(* CoDeSys 2.3.9.50 project: BallGame_with_PackMLandDriveFB_NT.pro *)
(* Libraries: TcBase.lib 14.5.09 11:14:08, TcSystem.lib 7.6.16 10:01:22, STANDARD.LIB 5.6.98 11:03:02 *)

(* Task configuration *)
TASK BallGame (PRIORITY := 1, INTERVAL := T#10ms);
	PRG_HMI();
	MAIN();
END_TASK
TASK Drive (PRIORITY := 0, INTERVAL := T#5ms);
	PRG_Drive_Link();
END_TASK
TASK Emergency (PRIORITY := 2, INTERVAL := T#5ms);
	PRG_SafetyProgram();
END_TASK

(* Global variable list: Global_Variables *)
VAR_GLOBAL
(* -------------INPUTS and OUTPUTS -------------------*)
(* See Global_Variables_TwinCAT and Global_Variables_CodeSys for
environment specific physical IOs *)

(*-----------------------TIMERS----------------------------*)
	TONMove_Ball_Delay		: TON;
	TONDrive_Delay			: TON;

(*-----------------------COUNTERS----------------------------*)
	CountBallsSortedMetal	: INT:=0;	(*Balls sorted: Metal*)
	CountBallsSortedWooden	: INT:=0;	(*Balls sorted: Wood*)
	CountBallsSortedYellow	: INT:=0;	(*Balls sorted: Wood, Yellow*)
	CountBallsSortedRed		: INT:=0;	(*Balls sorted: Wood, Red*)
	CountBallsSortedBlue	: INT:=0;	(*Balls sorted: Wood, Blue*)
	CountBallsSortedGarbage	: INT:=0;	(*Balls sorted: Unknown*)
	arrCountBallsOnTubes	: ARRAY [1..4] OF INT;	(*Balls on tubes: 1=lower, 2=middle, 3=upper, 4=garbage*)

(*-----------------------FUNCTION BLOCKS----------------*)
	fbDrive					: FB_DriveMovement2;		(*FB for executing the motion*)
	fbStateModel			: FB_StateModel_ST;		(*FB for executing state model*)

(* -------------HMI INPUTS (from HMI to PLC) -------------------*)
	bHMI_BtnStart			: BOOL;		(*Start button on HMI*)
	bHMI_BtnStartLight		: BOOL;		(*Start button Light on HMI*)
	bHMI_BtnStop			: BOOL;		(*Stop button on HMI*)
	bHMI_BtnStopLight		: BOOL;		(*Stop button Light on HMI*)
	bHMI_BtnReset			: BOOL;		(*Reset button on HMI*)
	bHMI_BtnAck		    	: BOOL;		(*Ack button on HMI*)

	HMI_uModeReq			: UINT := 3; (* Default to Sorting

(* -------------HMI OUTPUTS (from PLC to HMI) -------------------*)
	PLC_uModeCurrent		: UINT;		(*Current Mode*)
	PLC_uStateCurrent		: UINT;		(*Current State*)
	O_Light_BeaconRed		: BOOL;		(*Light beacon: Red*)

(*-----------------------OTHER GLOBAL VARS ----------------*)
	bInitCompleted			: BOOL; 	(*Init at Power Up *)
	iBatchSize				: INT := 1;	(*Default Batch Size *)
	iBatchRemaining			: INT;

END_VAR

VAR_GLOBAL CONSTANT
(*-----------------------Lift Position Constants----------------------------*)
	GPOS_LOADING			: WORD := 16#0A;	(*Drive to loading level*)
	GPOS_PIPE_LOW			: WORD := 16#0B;	(*Drive to lower pipe*)
	GPOS_PIPE_MID			: WORD := 16#0C;	(*Drive to middle pipe*)
	GPOS_PIPE_UP			: WORD := 16#0D;	(*Drive to upper pipe*)
	GPOS_GARBAGE			: WORD := 16#0E;	(*Drive to garbage pipe*)
	GPOS_COLOR_SEN			: WORD := 16#0F;	(*Drive to colour sensor*)

(*-----------------------Ball Type Constants----------------------------*)
	METAL					: BOOL := FALSE;
	WOODEN					: BOOL := TRUE;

(*-----------------------TIME Constants----------------------------*)
(*State Model *)
	T_IDLE_SHUTDOWN			: TIME := T#15s;
	T_START_DELAY			: TIME := T#2s;
(*Sorter*)
	T_CLEARING_BALL			: TIME := T#3s;
	T_BALL_DEBOUNCE			: TIME := T#500ms;
	T_LOADING_BALL			: TIME := T#1.5s;	(*Delay for ball to roll from Slot2 to Lifter*)
	T_ROLL_FROM_IND			: TIME := T#500ms;	(*Delay for ball to roll from Slot2 to Lifter*)
	T_REQ_DELAY				: TIME := T#500ms;
(*Drive/Lift*)
	T_RESET_DRIVE_TIME		: TIME := T#500ms;	(*Delay for ball to roll from Slot2 to Lifter*)
	T_DRIVE_DELAY			: TIME := T#2s;	(*Delay for drive to start movement*)
	T_POS_SETTLE_DELAY		: TIME := T#500ms;
	T_EJECTOR_DELAY			: TIME := T#500ms;
	T_COLOUR_SENSOR_DELAY	: TIME := T#1s;
(*Tubes *)
	T_TUBE_EMPTY_DELAY 		: TIME := T#3s;

END_VAR

(* Global variable list: Global_Variables_CodeSys *)
VAR_GLOBAL
(* -------------INPUTS-------------------*)
	ISensorOpt 			:BOOL;	(*Optical sensor - is ball present*)
	ISensorInd 			:BOOL;	(*Inductive sensor - is metal ball present*)
	IEmergencyClear 		:BOOL;	(*Emergency stop is cleared*)
	IRun 				:BOOL;	(*Run switch*)
	ILimitUp 				:BOOL;	(*Lift's limit switch is activated - Up*)
	ILimitLow 		 	:BOOL;	(*Lift's limit switch is activated - Low*)
	IGateClosedMid		:BOOL;	(*Pipe gate closed - Mid*)
	IGateClosedLow		:BOOL;	(*Pipe gate closed - Low*)
	ISorterGateClosed		:BOOL;	(*Sorter gate closed*)
	ISorterLiftUp			:BOOL;	(*Sorter lift at up position*)
	ISorterLiftDown		:BOOL;	(*Sorter lift at down position*)
	IPressureApplied		:BOOL;	(*Pressure is available for the system*)
	TEMP1				:BOOL;
	ISenColourYellow		:BOOL;	(*Colour sensor In1 - Yellow*)
	ISenColourBlue		:BOOL;	(*Colour sensor In2 - Blue*)
	ISenColourGreen		:BOOL;	(*Colour sensor In3 - Green*)
	ISenColourRed		:BOOL;	(*Colour sensor In4 - Red*)
	IDriveStatus 			:WORD;	(*From lift drive status information*)

(* -------------OUTPUTS-------------------*)
	OGateMid			:BOOL;	(*Valve: Open pipe gate - Mid*)
	OGateLow			:BOOL;	(*Valve: Open pipe gate - Low*)
	OSorterGate			:BOOL;	(*Valve: Open sorter gate*)
	OSorterLift			:BOOL;	(*Valve: Sorter lift up*)
	OEjector			:BOOL;	(*Ejector push ball out from lift*)
	ODriveControl 		:WORD;	(*To lift drive control information*)
END_VAR

(* Global variable list: Global_Variables_TwinCAT *)
VAR_GLOBAL
(* -------------INPUTS-------------------*)
	ISensorOpt 			AT %I*	:BOOL;	(*Optical sensor - is ball present*)
	ISensorInd 			AT %I*	:BOOL;	(*Inductive sensor - is metal ball present*)
	IEmergencyClear 	AT %I*	:BOOL;	(*Emergency stop is cleared*)
	IRun 				AT %I*	:BOOL;	(*Run switch*)
	ILimitUp 			AT %I*	:BOOL;	(*Lift's limit switch is activated - Up*)
	ILimitLow 			AT %I* 	:BOOL;	(*Lift's limit switch is activated - Low*)
	IGateClosedUp		AT %I* 	:BOOL;
	IGateClosedMid		AT %I*	:BOOL;	(*Pipe gate closed - Mid*)
	IGateClosedLow		AT %I*	:BOOL;	(*Pipe gate closed - Low*)
	ISorterGateClosed	AT %I*	:BOOL;	(*Sorter gate closed*)
	ISorterLiftUp		AT %I*	:BOOL;	(*Sorter lift at up position*)
	ISorterLiftDown		AT %I*	:BOOL;	(*Sorter lift at down position*)
	IPressureApplied	AT %I*	:BOOL;	(*Pressure is available for the system*)
	TEMP1				AT %I*	:BOOL;
	ISenColourYellow	AT %I*	:BOOL;	(*Colour sensor In1 - Yellow*)
	ISenColourBlue		AT %I*	:BOOL;	(*Colour sensor In2 - Blue*)
	ISenColourGreen		AT %I*	:BOOL;	(*Colour sensor In3 - Green*)
	ISenColourRed		AT %I*	:BOOL;	(*Colour sensor In4 - Red*)
	IDriveStatus 		AT %I*	:WORD;	(*From lift drive status information*)

(* -------------OUTPUTS-------------------*)
	OGateUp				AT %Q*	:BOOL;
	OGateMid			AT %Q*	:BOOL;	(*Valve: Open pipe gate - Mid*)
	OGateLow			AT %Q*	:BOOL;	(*Valve: Open pipe gate - Low*)
	OSorterGate			AT %Q*	:BOOL;	(*Valve: Open sorter gate*)
	OSorterLift			AT %Q*	:BOOL;	(*Valve: Sorter lift up*)
	OEjector			AT %Q*	:BOOL;	(*Ejector push ball out from lift*)
	ODriveControl 		AT %Q*	:WORD;	(*To lift drive control information*)

(* -------------HMI-------------------*)
	I_Btn_Reset		: BOOL;	(*Button: Reset*)
	I_Btn_Start		: BOOL;	(*Button: Start*)
	I_Btn_Stop		: BOOL;	(*Button: Stop*)
	I_Btn_EStop		: BOOL;	(*Button: Reset*)

(* -------------Drive-------------------*)
	bDriveEnabled 	: BOOL;

(* ------------ Manual Mode -------------*)
	bManualMode 	: BOOL := TRUE;
END_VAR

(* Global variable list: TwinCAT_Configuration *)
(* Generated automatically by TwinCAT - (read only) *)
VAR_CONFIG
	.ISensorOpt AT %IX0.0 : BOOL;	(*  ~ {LinkedWith:TIID^Device 4 (EL6731)^Box 2  (BK3110)^Term 2 (KL1002)^Channel 1^Input} *)
	.ISensorInd AT %IX0.1 : BOOL;	(*  ~ {LinkedWith:TIID^Device 4 (EL6731)^Box 2  (BK3110)^Term 2 (KL1002)^Channel 2^Input} *)
	.IEmergencyClear AT %IX0.2 : BOOL;	(*  ~ {LinkedWith:TIID^Device 4 (EL6731)^Box 2  (BK3110)^Term 3 (KL1002)^Channel 1^Input} *)
	.IRun AT %IX0.3 : BOOL;	(*  ~ {LinkedWith:TIID^Device 4 (EL6731)^Box 2  (BK3110)^Term 3 (KL1002)^Channel 2^Input} *)
	.ILimitUp AT %IX0.4 : BOOL;	(*  ~ {LinkedWith:TIID^Device 4 (EL6731)^Box 2  (BK3110)^Term 4 (KL1002)^Channel 1^Input} *)
	.ILimitLow AT %IX0.5 : BOOL;	(*  ~ {LinkedWith:TIID^Device 4 (EL6731)^Box 2  (BK3110)^Term 4 (KL1002)^Channel 2^Input} *)
	.IGateClosedUp AT %IX8.0 : BOOL;
	.IGateClosedMid AT %IX0.7 : BOOL;	(*  ~ {LinkedWith:TIID^Device 4 (EL6731)^Box 2  (BK3110)^Term 5 (KL1104)^Channel 2^Input} *)
	.IGateClosedLow AT %IX1.0 : BOOL;	(*  ~ {LinkedWith:TIID^Device 4 (EL6731)^Box 2  (BK3110)^Term 5 (KL1104)^Channel 3^Input} *)
	.ISorterGateClosed AT %IX1.1 : BOOL;	(*  ~ {LinkedWith:TIID^Device 4 (EL6731)^Box 2  (BK3110)^Term 5 (KL1104)^Channel 4^Input} *)
	.ISorterLiftUp AT %IX1.2 : BOOL;	(*  ~ {LinkedWith:TIID^Device 4 (EL6731)^Box 2  (BK3110)^Term 6 (KL1104)^Channel 1^Input} *)
	.ISorterLiftDown AT %IX1.3 : BOOL;	(*  ~ {LinkedWith:TIID^Device 4 (EL6731)^Box 2  (BK3110)^Term 6 (KL1104)^Channel 2^Input} *)
	.IPressureApplied AT %IX1.4 : BOOL;	(*  ~ {LinkedWith:TIID^Device 4 (EL6731)^Box 2  (BK3110)^Term 6 (KL1104)^Channel 3^Input} *)
	.TEMP1 AT %IX1.5 : BOOL;	(*  ~ {LinkedWith:TIID^Device 4 (EL6731)^Box 2  (BK3110)^Term 6 (KL1104)^Channel 4^Input} *)
	.ISenColourYellow AT %IX1.6 : BOOL;	(*  ~ {LinkedWith:TIID^Device 4 (EL6731)^Box 2  (BK3110)^Term 7 (KL1104)^Channel 1^Input} *)
	.ISenColourBlue AT %IX1.7 : BOOL;	(*  ~ {LinkedWith:TIID^Device 4 (EL6731)^Box 2  (BK3110)^Term 7 (KL1104)^Channel 2^Input} *)
	.ISenColourGreen AT %IX2.0 : BOOL;	(*  ~ {LinkedWith:TIID^Device 4 (EL6731)^Box 2  (BK3110)^Term 7 (KL1104)^Channel 3^Input} *)
	.ISenColourRed AT %IX2.1 : BOOL;	(*  ~ {LinkedWith:TIID^Device 4 (EL6731)^Box 2  (BK3110)^Term 7 (KL1104)^Channel 4^Input} *)
	.IDriveStatus AT %IB4 : WORD;	(*  ~ {LinkedWith:TIID^Device 4 (EL6731)^Box 5 (DKC03)^DKC03 mit LSPM2^Inputs^DKC03 mit LSPM2_0_0} *)
	.OGateUp AT %QX4.0 : BOOL;
	.OGateMid AT %QX0.1 : BOOL;	(*  ~ {LinkedWith:TIID^Device 4 (EL6731)^Box 2  (BK3110)^Term 8 (KL2114)^Channel 2^Output} *)
	.OGateLow AT %QX0.2 : BOOL;	(*  ~ {LinkedWith:TIID^Device 4 (EL6731)^Box 2  (BK3110)^Term 8 (KL2114)^Channel 3^Output} *)
	.OSorterGate AT %QX0.3 : BOOL;	(*  ~ {LinkedWith:TIID^Device 4 (EL6731)^Box 2  (BK3110)^Term 8 (KL2114)^Channel 4^Output} *)
	.OSorterLift AT %QX0.4 : BOOL;	(*  ~ {LinkedWith:TIID^Device 4 (EL6731)^Box 2  (BK3110)^Term 9 (KL2114)^Channel 1^Output} *)
	.OEjector AT %QX0.5 : BOOL;	(*  ~ {LinkedWith:TIID^Device 4 (EL6731)^Box 2  (BK3110)^Term 9 (KL2114)^Channel 2^Output} *)
	.ODriveControl AT %QB2 : WORD;	(*  ~ {LinkedWith:TIID^Device 4 (EL6731)^Box 5 (DKC03)^DKC03 mit LSPM2^Outputs^DKC03 mit LSPM2_1_0} *)
END_VAR

(* Data type *)
TYPE E_BallColour :
(
	NoColour := 0,
	Yellow := 1,
	Blue := 2,
	Red := 3
);
END_TYPE

(* Data type *)
TYPE E_ModeCtrl :
(
	eMode_undefined := 0,
	eMode_Automatic :=1,
	eMode_XXX :=2,
	eMode_Manual :=99,
	eMode_Sorting :=3,
	eMode_Emptying :=4
);
END_TYPE

(* Data type *)
TYPE E_ModeProc :
(*Procedural control modes. Can be changed in any state*)
(
	eModeProc_undefined := 0,
	eModeProc_Automatic :=1,
	eModeProc_SemiAutomatic :=2,
	eModeProc_Manual :=3
);
END_TYPE

(* Data type *)
TYPE E_State :
(
	eSt_Aborting :=0,
	eSt_Aborted,
	eSt_Clearing,
	eSt_Stopped,
	eSt_Stopping,
	eSt_Resetting,
	eSt_Idle,
	eSt_Starting,
	eSt_Execute,
	eSt_Suspending,
	eSt_Suspended,
	eSt_Unsuspending,
	eSt_Holding,
	eSt_Held,
	eSt_UnHolding,
	eSt_Completing,
	eSt_Completed
);
END_TYPE

(* POU PRG_HMI, ST *)
PROGRAM PRG_HMI
VAR_INPUT
	(*HMI Buttons*)
	bBtnResetCounters	: BOOL;	(*Button Reset counters*)
	bBtnEmptyPipes		: BOOL;	(*Button Empty Pipes*)
END_VAR
VAR

	(*Variables for Lift visualisation*)
	iSorterLiftPos	: INT;		(*Position of Sorter Lift cylinder*)
	iLiftPos		: INT;		(*Position of the lift*)
	wTargetPos	: INT;		(*Current target position of the lift*)
	bBall_InLift	: BOOL;		(*Is there a ball in lift*)

	(*internal variables*)
	RS_Ball_InLift	: RS;		(*Flip-flop for ball in the lift*)
	i: INT := 0;		(*Counter*)
	ii: INT := 0;
	SR_EmptyTubes	: SR;


END_VAR
(*Producing blinking signal*)
PRG_Blinking();

(*Sorter lift position calculus*)
IF OSorterLift AND (iSorterLiftPos < 30) THEN
	iSorterLiftPos := iSorterLiftPos +10;
END_IF;
IF NOT OSorterLift AND (iSorterLiftPos > 0) THEN
	iSorterLiftPos := iSorterLiftPos - 10;
END_IF;

(*Lift position calculus*)
CASE fbDrive.wDestination OF
GPOS_PIPE_UP:		(*Go to Pipe Up*)
	wTargetPos:=375;
GPOS_PIPE_MID:	(*Go to Pipe Mid*)
	wTargetPos:=275;
GPOS_COLOR_SEN:	(*Go to Colour sensor*)
	wTargetPos:=220;
GPOS_PIPE_LOW:	(*Go to Pipe Low*)
	wTargetPos:=175;
GPOS_GARBAGE:	(*Go to garbage position*)
	wTargetPos:=110;
GPOS_LOADING:	(*Go to loading position*)
	wTargetPos:=20;
ELSE
	wTargetPos:=0;
END_CASE;

ii := ii + 1;
(*Drive lift*)
IF( ii MOD 3 = 0) THEN
	IF iLiftPos > wTargetPos THEN	(*Lift is higher than target*)
		iLiftPos := iLiftPos - 1;	 (*Go down*)
	ELSIF iLiftPos < wTargetPos THEN	(*Lift is lower than target*)
		iLiftPos := iLiftPos + 1;	 (*Go up*)
	END_IF;
END_IF;

(*Is there a ball in the lift*)
RS_Ball_InLift(
	SET:= (iLiftPos=20 AND OSorterGate),
	RESET1:=OEjector ,
	Q1=>bBall_InLift );

(* ---------------------------------- Button handlers ---------------------------------- *)
(*Button Empty Pipes*)
SR_EmptyTubes (
	SET1:= bBtnEmptyPipes,
	RESET:=,
	Q1=> );
IF SR_EmptyTubes.Q1 THEN
	PRG_EmptyTubes(bExecute:= TRUE, bDone:= );
	SR_EmptyTubes.RESET := FALSE;
	IF PRG_EmptyTubes.bDone THEN
		PRG_EmptyTubes(bExecute:= FALSE);
		SR_EmptyTubes.RESET := TRUE;
	END_IF
END_IF

(*Button Reset coutners*)
IF bBtnResetCounters THEN
	CountBallsSortedMetal := 0;
	CountBallsSortedWooden := 0;
	CountBallsSortedYellow := 0;
	CountBallsSortedBlue := 0;
	CountBallsSortedRed := 0;
	CountBallsSortedGarbage := 0;
	FOR i := 1 TO 3 DO
		arrCountBallsOnTubes[i] := 0;
	END_FOR;
END_IF;
END_PROGRAM

(* POU Background Programs/PRG_Blinking, ST *)
PROGRAM PRG_Blinking
(*Supporting caluculations: Blinking signals
Author: 	Niko Siltala, niko.siltala@tut.fi
Date: 	2014-01-01*)

VAR_OUTPUT
	bSign4Hz	:BOOL;				(*4 Hz (240krt/min) taajudella vaihteleva signaali*)
	bSign2Hz	:BOOL;				(*2 Hz (120krt/min) taajudella vaihteleva signaali*)
	bSign1Hz	:BOOL;				(*1 Hz (60krt/min) taajudella vaihteleva signaali*)
	bSign0_5Hz	:BOOL;				(*0,5 Hz (30krt/min) taajudella vaihteleva signaali*)
END_VAR
VAR
	bInitDone	: BOOL	:=FALSE;		(*Ohjelman initialisointi*)
	TP_Delay	: TP;					(*Nopein taajuus / 2 tuottaja*)
	bBaseHz	: BOOL	:=FALSE;		(*Nopein taajuus/2*)
	iBaseHz		: UINT	:=4;			(*Base taajuus (Hz)*)
	RTRIG_2Hz_Sign 	: R_TRIG;		(*2Hz signaalin generointi*)
	RTRIG_1Hz_Sign 	: R_TRIG;		(*1Hz signaalin generointi*)
	RTRIG_0_5Hz_Sign	: R_TRIG;	(*0,5Hz signaalin generointi*)
	tBaseTaajuus	:TIME;			(*Base vilkutuksen timerin arvo. f/2*)
	fPLC_CYCLE_TIME	: LREAL;		(*PLC:n cycli aika. Sekunttia*)
END_VAR
(*Ohjelman initialisoinnit - Suoritetaan vain kertaalleen*)
IF NOT bInitDone THEN
	fPLC_CYCLE_TIME := UDINT_TO_LREAL(SystemTaskInfoArr[1].cycleTime) / 10E6;
	(*Base Vilkkusignaalien tuottaminen*)
	(* 250ms - 1* cykliaika(20ms)*)
	tBaseTaajuus := LREAL_TO_TIME( ( (1/ UINT_TO_LREAL(iBaseHz) / 2 ) - 1 * fPLC_CYCLE_TIME ) * 1000);
	bInitDone := TRUE;
END_IF;


(*Base signaalin genrointi*)
TP_Delay(IN:=NOT TP_Delay.Q , PT:=tBaseTaajuus);
IF NOT TP_Delay.Q THEN
	bBaseHz := NOT bBaseHz;
	bSign4Hz:= bBaseHz;
END_IF;

(*2Hz signaalin genrointi*)
RTRIG_2Hz_Sign(CLK:=bSign4Hz);
IF RTRIG_2Hz_Sign.Q THEN
	bSign2Hz:=NOT bSign2Hz;
END_IF;

(*1Hz signaalin genrointi*)
RTRIG_1Hz_Sign(CLK:=bSign2Hz);
IF RTRIG_1Hz_Sign.Q THEN
	bSign1Hz:=NOT bSign1Hz;
END_IF;

(*0,5 Hz signaalin generointi*)
RTRIG_0_5Hz_Sign(CLK:=bSign1Hz);
IF (RTRIG_0_5Hz_Sign.Q) THEN
	bSign0_5Hz:= NOT bSign0_5Hz;
END_IF;
END_PROGRAM

(* POU Processes/PRG_EmptyTubes, SFC *)
(* This Program performs the emptying of the tubes in a set sequence
to prevent jamming. Used in User mode: Emptying
Author: Nicolas Trimborn, nicolas.trimborn@tuni.fi
Date: 	2020-03-01*)

PROGRAM PRG_EmptyTubes
VAR_INPUT
	bExecute	: BOOL;
END_VAR
VAR_INPUT
	bDone		: BOOL;
	bStopOk		: BOOL;
END_VAR
VAR
	fbDelay		:FB_Wait;
END_VAR
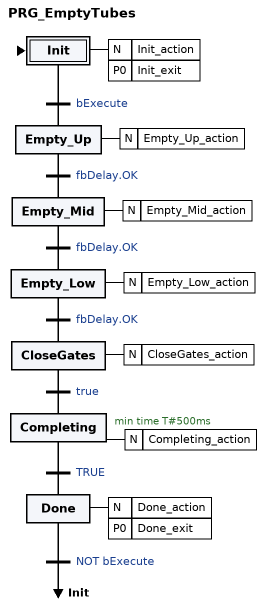
INITIAL_STEP Init:
	Init_action(N);
	Init_exit(P0);
END_STEP
TRANSITION FROM Init TO Empty_Up := bExecute;
END_TRANSITION
STEP Empty_Up:
	Empty_Up_action(N);
END_STEP
TRANSITION FROM Empty_Up TO Empty_Mid := fbDelay.OK;
END_TRANSITION
STEP Empty_Mid:
	Empty_Mid_action(N);
END_STEP
TRANSITION FROM Empty_Mid TO Empty_Low := fbDelay.OK;
END_TRANSITION
STEP Empty_Low:
	Empty_Low_action(N);
END_STEP
TRANSITION FROM Empty_Low TO CloseGates := fbDelay.OK;
END_TRANSITION
STEP CloseGates:
	CloseGates_action(N);
END_STEP
TRANSITION FROM CloseGates TO Completing := true;
END_TRANSITION
STEP Completing: (* min time T#500ms *)
	Completing_action(N);
END_STEP
TRANSITION FROM Completing TO Done := TRUE;
END_TRANSITION
STEP Done:
	Done_action(N);
	Done_exit(P0);
END_STEP
TRANSITION FROM Done TO Init := NOT bExecute;
END_TRANSITION

ACTION Init_action:
bStopOk := TRUE;
END_ACTION

ACTION Init_exit:
(* Sequence is executing, Reset progress flags *)
bDone 	:= FALSE;
bStopOk := FALSE;
END_ACTION

ACTION Empty_Up_action:
fbDelay(IN_TIME:=T_TUBE_EMPTY_DELAY);
OGateUp := TRUE;
END_ACTION

ACTION Empty_Mid_action:
fbDelay(IN_TIME:=T_TUBE_EMPTY_DELAY);
OGateMid := TRUE;
END_ACTION

ACTION Empty_Low_action:
fbDelay(IN_TIME:=T_TUBE_EMPTY_DELAY);
OGateLow := TRUE;
END_ACTION

ACTION CloseGates_action:
OGateLow := FALSE;
OGateMid := FALSE;
OGateUp  := FALSE;
END_ACTION

ACTION Completing_action:
fbStateModel.bComplete := TRUE;
END_ACTION

ACTION Done_action:
(* Sequence Completed, set progress flags *)
bDone := TRUE;
bStopOk := TRUE;
fbStateModel.bSC := TRUE;
END_ACTION

ACTION Done_exit:
bDone := FALSE;
END_ACTION
END_PROGRAM

(* POU FBs/FB_Wait, ST *)
FUNCTION_BLOCK FB_Wait
(*Waits the given time and sets output after timer has run till end. When called again timer restarts.
Author: 	Niko Siltala, niko.siltala@tut.fi
Date: 	2014-01-01*)
VAR_INPUT
	IN_TIME	:TIME;		(*Time to wait*)
END_VAR
VAR_OUTPUT
	OK 		: BOOL:=FALSE;	(*Gets true after wait time has expired*)
END_VAR
VAR
	Timer	: TP;
	Falling	: F_TRIG;
END_VAR
IF Timer.Q=TRUE THEN
	(*Call timer block when pulse timer is counting*)
	Timer;
ELSE
	(*Timer has espired. Start it again*)
	Timer(IN:=FALSE);
	Timer(PT:=IN_TIME);
	Timer(IN:=TRUE);
END_IF;
(*Set output. True if timer has expired*)
OK:=NOT Timer.Q;
END_FUNCTION_BLOCK

(* POU MAIN, ST *)
(* Main performs Implements PackML model to control the execution of the application
used to coordinate machine operation. 
User modes are:
 - Sorting
 - Emptying
PRG_Safety is running as a separate process to monitor the Estop and limit switches
to shut down drive regardless of other program logic.
Author: Nicolas Trimborn, nicolas.trimborn@tuni.fi
Date: 	2020-03-01*)

PROGRAM MAIN

VAR
	runTrigger			: R_TRIG;
	stopTrigger			: F_TRIG;
	tonStarting			: TON;	(* Start timer used to provide notification machine is starting *)
	rsEmergencyClear	: RS;	(*RS - flip-flop for Emergency clear info*)
	fbPipeUp    		: FB_Pipe;
	fbPipeMid   		: FB_Pipe;
	fbPipeLow   		: FB_Pipe;
	fbDelay				: FB_Wait;
END_VAR
(* ****** Section 1: Initialisations and default values. Initial conditions for variables on every PLC cycle*)
(*Default values*)
fbStateModel.bSC := FALSE;
runTrigger(CLK := IRun); (* finds the counting up events *)
stopTrigger(CLK := IRun); (* finds the clear commands *)

(*System resets*)

(* ****** Section 2: Actions in your program without considering the Control Mode. I.e. actions are performed same way indenpendent on
current Control Mode selection.*)
(*Mode independent state actions. Change / Add / Remove states according your need*)
CASE fbStateModel.eState OF
	eSt_Aborting: (* Handles aborting action such as E-Stop, Limit Switches and Pressure loss *)
		actAborting;
		fbStateModel.bSC := TRUE;		(*MODIFY*)
	eSt_Clearing:
		fbDrive(bReset := TRUE);
		fbDelay(IN_TIME:= T_RESET_DRIVE_TIME, OK=> );
		IF fbDelay.OK THEN
			fbDrive(bReset := FALSE);
			fbStateModel.bSC := TRUE;
		END_IF
	eSt_Resetting:
		tonStarting(IN:=FALSE , PT:= , Q=> , ET=> );	(*MODIFY*)
		fbStateModel.bComplete  := FALSE;
		fbStateModel.bSC := TRUE;
	eSt_Starting:
		(* Reset Program Reset Flags *)
		PRG_Initialisation(bReset := FALSE);
		PRG_Sorting.bReset := FALSE;
		PRG_HMI.bBtnResetCounters := FALSE;
		(* Starting Sequence,  Need to check that pressure is avalible and emergency is clear *)
		IF NOT bInitCompleted THEN (* Initial Startup - Perform Initialisation *)
			PRG_Initialisation(bExecute:= TRUE, bReset := FALSE );
		ELSE (* Init Not Required, Start after 2s delay *)
			fbDrive(bEnable:= TRUE, bStart := TRUE);
			IF fbDrive.bHomingDone THEN
				tonStarting(IN:=TRUE , PT:=T_START_DELAY , Q=> , ET=> );
				IF tonStarting.Q THEN
					fbStateModel.bSC := TRUE;
				END_IF
			END_IF
		END_IF
	
		IF PRG_Initialisation.bDone THEN (*Initialisation Program Is Done *)
			(*Reset Init Program and set bInitComplete flag to indicate Init Performed on Power Up*)
			PRG_Initialisation(bReset:= , bExecute:= FALSE , bDone=> );
			bInitCompleted := TRUE;
		END_IF
	eSt_Holding:
		fbStateModel.bSC := TRUE;		(*MODIFY*)
	eSt_UnHolding:
		fbStateModel.bSC := TRUE;		(*MODIFY*)
	eSt_Suspending:
		fbStateModel.bSC := TRUE;		(*MODIFY*)
	eSt_Unsuspending:
		fbStateModel.bSC := TRUE;		(*MODIFY*)
END_CASE;

(* ****** Section 3: Actions in your program which are Control Mode specific. Two nested case structures where outer one selects the
control mode and inner the PackML state. In order to avoid conflicts, it would be better to process each PackML state either in Section 2 
or Section 3, but not in both. *)
(*Execution mode related state actions. Change / Add / Remove mode and states according your need*)
CASE fbStateModel.eMode OF
	(* ********************* MODE: Emptying******************************************************* *)
	eMode_Emptying:
		(* ****** Section 3.1: PackML state based processing actions when Control Mode is Emptying.*)
		CASE fbStateModel.eState OF
			eSt_Stopping: (*Ensure sequence completeded before stopping, Nice Stop*)
				PRG_EmptyTubes(bExecute:= FALSE, bDone:= , bStopOk:= );
				IF PRG_EmptyTubes.bStopOk THEN
					fbStateModel.bSC := TRUE;
				END_IF
			eSt_Completed:
				fbStateModel.bComplete  := FALSE;
				PRG_EmptyTubes(bExecute := FALSE);
				PRG_HMI.bBtnResetCounters := TRUE;
		END_CASE;

		IF  (fbStateModel.eState>eSt_Starting) AND (fbStateModel.eState<=eSt_Completing) THEN (*State is equal or above Stopped*)
			(*Make here the actions / calls Good place to start with is PRG_Sorting (PRG)*)
			PRG_EmptyTubes(bExecute:= TRUE, bDone:= , bStopOk:= );

		END_IF;

	(* ********************* MODE: Manual ******************************************************* *)
	eMode_Manual:
		CASE fbStateModel.eState OF
		eSt_Stopping:
			;
		eSt_Execute:
			;
		END_CASE;


	(* ********************* MODE: Sorting ****************************************************** *)
	eMode_Sorting:
		(* ****** Section 3.2: PackML state based processing actions when Control Mode is Sorting.*)
		CASE fbStateModel.eState OF
		(*
		eSt_Idle:
			(* Reset Start Counter and bComplete Flag
			tonStarting(IN:=FALSE , PT:= , Q=> , ET=> );
			fbStateModel.bComplete  := FALSE;
			fbStateModel.bSC 		:= TRUE; *)
		eSt_Stopping:
			PRG_Sorting(bExecute:= FALSE, bDone:= , bStopOk:= );
			IF PRG_Sorting.bStopOk THEN
				fbStateModel.bSC := TRUE;
			END_IF
		eSt_Completed:
			fbStateModel.bComplete := FALSE;
			IF fbStateModel.bAck_Completed OR bHMI_BtnAck THEN
				PRG_HMI.bBtnResetCounters := TRUE;
				PRG_Sorting.bReset := TRUE;
			END_IF
			;
		END_CASE; (*fbStateModel.eState *)

	(* ****** Section 4: Grouping PackML states for calling Programs or FB instances.
	This is to avoid repetition inside above case structure in Section 3. With IF clause setting lower (and upper) state limits we can filter out the states when we want to call 
	specific programs. The order of states is defined in Tab:Data types > E_PackMLState. eSt_Aborting is lowest and eSt_Completed is highest.
	Here we filter calling programs, only when we are in higher states than Stopped. 
	This can be pulled out as completely separated section, like in PackML_StateModel_v2-2.pro project. There is inside IF again CASE which process each Control Mode separately.*)
	(*Execution part. Making calls for program if we are on states above Stopped*)
		(*If we are between specific states, make some action or program call*)
			(*IF  (fbStateModel.eState>eSt_Starting) AND (fbStateModel.eState<=eSt_Completing) THEN*)
		IF  (fbStateModel.eState>eSt_Starting) AND (fbStateModel.eState<=eSt_Completing) THEN (*State is equal or above Stopped*)
			(*Make here the actions / calls Good place to start with is PRG_Sorting (PRG)*)
			PRG_Sorting(bExecute:= TRUE , bReset:= , bDone=> , bStopOk=>, iBatchSize := iBatchSize );
		END_IF;

	(* ********************* End of MODE: Sorting******************************************************* *)


	(* fbStateModel.eMode, MODE: UNKNOWN*)
	ELSE	(*Error*)
		; (*TODO*)
END_CASE;

(* ****** Section 5: Calling the fbStateModel instance.
Here the instance of state model is called and all triggering inputs are set, but bSC (State Completed), which you control in your programs. 
This is indication that your program has  finished certain stage.
- Pay attention where the instance fbStateModel is defined. Do you do it in global variables or e.g. here in PRG_MAIN? Important is to use the 
same instance in all places, so that machine state is unique and shared. Remember, if you have multiple definitions, the PRG_MAIN "hides" 
the global one, and might lead to problems elswhere, when you think you are using the same instance, but actually are not. 
- In case you are using the PackML visualisation (VC_PackMLStates), make sure you connect its placeholder to the very same PackML FB instance.
- The Mask for wIgnoreState is created as following. I use binary base for the value(2#). The lowest bit in the mask corresponds the eSt_Aborting
 in E_PackMLState. The next is eSt_Aborted, and so on. Specific state is ignored and jumped over when it is masked out i.e. ignored by having 1 
in that position. Note that implementation allows this only for selected states. See FB_PackMLStateModel_ST code for further details.*)
(*Calling & Updating the state model*)
(*TODO: Evaluate and change all input conditions according your application needs*)
fbStateModel(
	bResetFB:= ,
	eModeReq:= HMI_uModeReq,
	wIgnoreState := 2#1000000,		(*TODO: Which states should be ignodered. Default: 2#000000 or 2#100000. The latter is ignoring Resetting state*)
	bSC:= ,			(*Must not be assigned ANY variable, because fb input is directly operated!!!*)
	bAbort:= NOT IEmergencyClear OR NOT IPressureApplied OR ILimitLow OR ILimitUp,
	bClear:= IEmergencyClear,
	bReset:= runTrigger.Q OR bHMI_BtnReset OR bHMI_BtnStart,
	bStart:= runTrigger.Q OR bHMI_BtnStart,
	bHold:= ,
	bUn_Hold:= ,
	bSuspend:= ,
	bUn_Suspend:= ,
	bStop:= bHMI_BtnStop OR stopTrigger.Q,
	bComplete:= ,
	bAck_Completed:= bHMI_BtnAck OR bHMI_BtnReset ,
	eMode=> PLC_uModeCurrent,
	eState=> PLC_uStateCurrent);

(* ****** Section 6: Here we update all outputs according the current state of our PackML model. This allows us to process the in single location.
The control of outputs is bind to state, not e.g. to inputs. The inputs are the one driving the PackML model forward. Again CASE structure can be used.*)
(*Call for HMI and UI update*)
(*PRG_Drive_Link()*);
HMI_and_UI_Update;
END_PROGRAM
ACTION actAborting:
(*PRG_Sorting(bReset:=TRUE , bExecute:= FALSE);*)
(*bInitCompleted := FALSE;*)
fbDrive(bEnable:= FALSE );
;
END_ACTION
ACTION HMI_and_UI_Update:
(*Simulate emergency stop circuitry
rsEmergencyClear(
	SET:= I_Btn_Reset,
	RESET1:= I_Btn_EStop ,
	Q1=> IEmergencyClear);
*)

(*HMI Update*)
PRG_Blinking (bSign4Hz=> , bSign2Hz=> , bSign1Hz=> , bSign0_5Hz=> );
PRG_Sorting.actCountBallsProcessed;
(*iBatchRemaining := iBatchSize - PRG_AutoSort.iBallsProcessed;*)

(*Init values*)
O_Light_BeaconRed := FALSE;
fbPipeLow(str_PipeName:= 'Metal', i_arrCountBallsIndex := 1, I_GateClosed := IGateClosedLow );
fbPipeMid(str_PipeName:= 'Wood, Blue' , i_arrCountBallsIndex := 2, I_GateClosed := IGateClosedMid );
fbPipeUp(str_PipeName:= 'Wood, Yellow', i_arrCountBallsIndex := 3, I_GateClosed := IGateClosedUp );

(*OLight_Start :=  (fbStateModel.eState >= eSt_Resetting) AND (fbStateModel.eState < eSt_Completed);*)
CASE fbStateModel.eState OF
eSt_Aborting, eSt_Aborted:
	O_Light_BeaconRed := PRG_Blinking.bSign1Hz;
	bHMI_BtnStartLight:= FALSE;
	bHMI_BtnStopLight := PRG_Blinking.bSign1Hz;
eSt_Clearing:
	O_Light_BeaconRed := PRG_Blinking.bSign0_5Hz;
	bHMI_BtnStopLight := PRG_Blinking.bSign0_5Hz;
eSt_Stopped, eSt_Completed:
	O_Light_BeaconRed := TRUE;
	bHMI_BtnStartLight:= FALSE;
	bHMI_BtnStopLight := TRUE;
eSt_Starting:
	bHMI_BtnStartLight := PRG_Blinking.bSign0_5Hz;
	bHMI_BtnStopLight := FALSE;
eSt_Stopping:
	bHMI_BtnStartLight := PRG_Blinking.bSign1Hz;
	bHMI_BtnStopLight := TRUE;
eSt_Execute:
	bHMI_BtnStartLight := TRUE;
	bHMI_BtnStopLight := FALSE;
	;
END_CASE;
END_ACTION

(* POU FBs/FB_Pipe, SFC *)
FUNCTION_BLOCK FB_Pipe
VAR_INPUT
	bReset					: BOOL;	(*Reset Request*)
	str_PipeName			: STRING;
	i_arrCountBallsIndex	: INT;
	I_GateClosed			: BOOL;
END_VAR
VAR_OUTPUT

END_VAR
VAR
	iBallCount  : INT := 0;
	tBallDelay	: TIME := T#1s;
	fbDelay		: FB_Wait;
	bLocalReset	: BOOL;	(*Performs local reset*)
	SFCReset 	: BOOL;	(*Resets the execution of SFC to init once this SFCFlag is set true *)
END_VAR
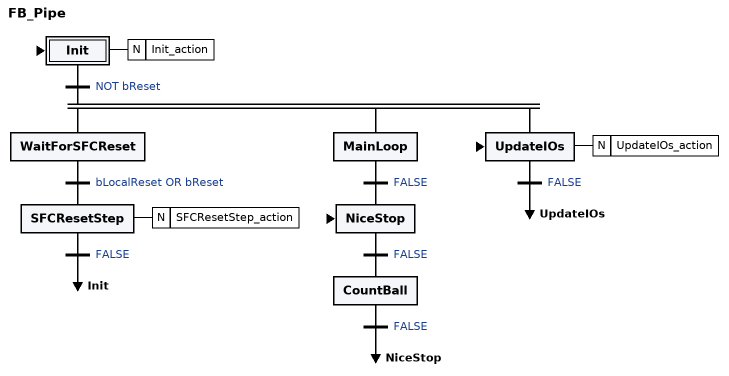
INITIAL_STEP Init:
	Init_action(N);
END_STEP
TRANSITION FROM Init TO (WaitForSFCReset, MainLoop, UpdateIOs) := NOT bReset;
END_TRANSITION
STEP WaitForSFCReset:
END_STEP
TRANSITION FROM WaitForSFCReset TO SFCResetStep := bLocalReset OR bReset;
END_TRANSITION
STEP MainLoop:
END_STEP
TRANSITION FROM MainLoop TO NiceStop := FALSE;
END_TRANSITION
STEP NiceStop:
END_STEP
TRANSITION FROM NiceStop TO CountBall := FALSE;
END_TRANSITION
STEP CountBall:
END_STEP
TRANSITION FROM CountBall TO NiceStop := FALSE;
END_TRANSITION
STEP UpdateIOs:
	UpdateIOs_action(N);
END_STEP
TRANSITION FROM UpdateIOs TO UpdateIOs := FALSE;
END_TRANSITION
STEP SFCResetStep:
	SFCResetStep_action(N);
END_STEP
TRANSITION FROM SFCResetStep TO Init := FALSE;
END_TRANSITION

ACTION Init_action:
SFCReset := FALSE;
bLocalReset	:= FALSE;
END_ACTION

ACTION UpdateIOs_action:
iBallCount := arrCountBallsOnTubes[i_arrCountBallsIndex];
END_ACTION

ACTION SFCResetStep_action:
SFCReset := TRUE;
END_ACTION
END_FUNCTION_BLOCK

(* POU Processes/PRG_Initialisation, SFC *)
(* This Program performs the initialising of the sorting machine to ensure it
enters a know state before sorting begins.  
- Clears sorter lift to ensure any balls left drop to lift
- Close Pipe Gates
- Home Lift and take any balls to garbage chute before returning to loading pos.
Author: Nicolas Trimborn, nicolas.trimborn@tuni.fi
Date: 	2020-03-01*)

PROGRAM PRG_Initialisation
(*Template program for system initialisation*)
VAR_INPUT
	bReset			: BOOL := FALSE;(*Reseting the SFC*)
	bExecute		: BOOL;			(*Executes PRG*)
END_VAR
VAR_OUTPUT
	bDone			: BOOL;			(*Program operations done*)
END_VAR
VAR
(* -------------INTERNAL-------------------*)
	tonMoveDelay	: TON;
	tonBallClearing	: TON;
	fbDelay			: FB_Wait;

	bSorterLiftClear: BOOL:=FALSE;
	bGatesClosed	: BOOL:=FALSE;
	bActuRetracted	: BOOL:=FALSE;
	bDriveAtLoading	: BOOL:=FALSE;
	bDriveReady		: BOOL:=FALSE;

(*System variables. See SFC-flags: http://infosys.beckhoff.com/content/1033/tcplccontrol/html/tcplcctrl_editorsfc.htm?id=24319#SFC-Flags*)
	SFCReset		: BOOL := FALSE;	(*For reseting the SFC*)
END_VAR
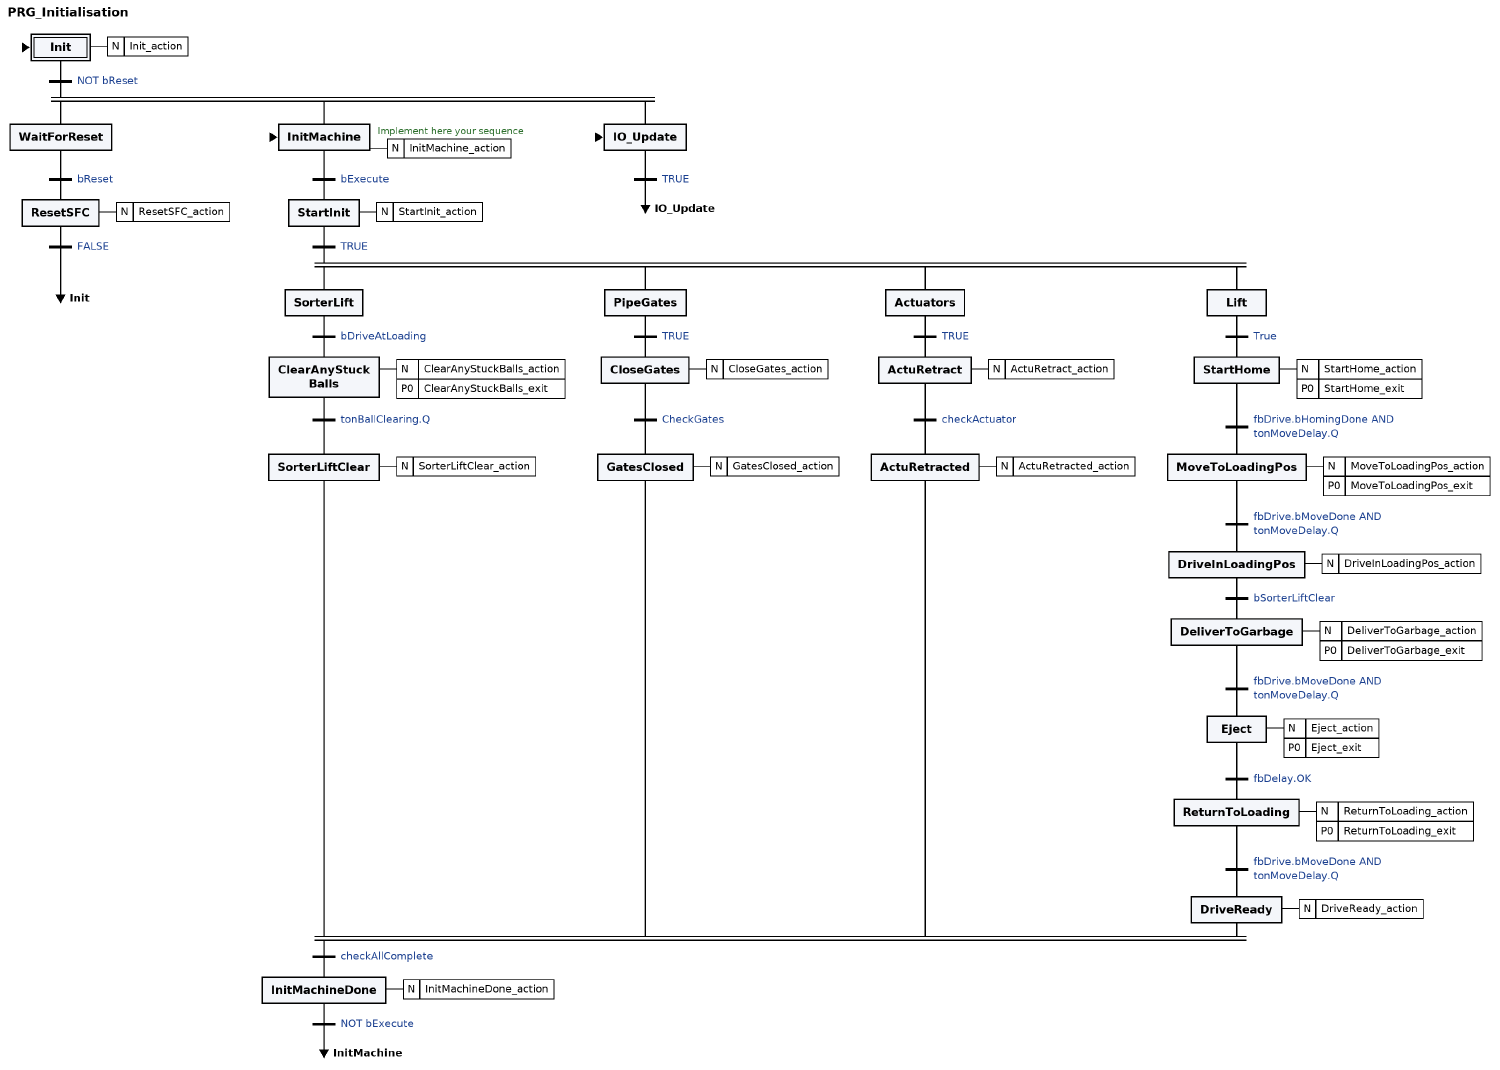
INITIAL_STEP Init:
	Init_action(N);
END_STEP
TRANSITION FROM Init TO (WaitForReset, InitMachine, IO_Update) := NOT bReset;
END_TRANSITION
STEP WaitForReset:
END_STEP
TRANSITION FROM WaitForReset TO ResetSFC := bReset;
END_TRANSITION
STEP InitMachine: (* Implement here your sequence *)
	InitMachine_action(N);
END_STEP
TRANSITION FROM InitMachine TO StartInit := bExecute;
END_TRANSITION
STEP StartInit:
	StartInit_action(N);
END_STEP
TRANSITION FROM StartInit TO (SorterLift, PipeGates, Actuators, Lift) := TRUE;
END_TRANSITION
STEP SorterLift:
END_STEP
TRANSITION FROM SorterLift TO ClearAnyStuckBalls := bDriveAtLoading;
END_TRANSITION
STEP ClearAnyStuckBalls:
	ClearAnyStuckBalls_action(N);
	ClearAnyStuckBalls_exit(P0);
END_STEP
TRANSITION FROM ClearAnyStuckBalls TO SorterLiftClear := tonBallClearing.Q;
END_TRANSITION
STEP SorterLiftClear:
	SorterLiftClear_action(N);
END_STEP
STEP PipeGates:
END_STEP
TRANSITION FROM PipeGates TO CloseGates := TRUE;
END_TRANSITION
STEP CloseGates:
	CloseGates_action(N);
END_STEP
TRANSITION FROM CloseGates TO GatesClosed := CheckGates;
END_TRANSITION
STEP GatesClosed:
	GatesClosed_action(N);
END_STEP
STEP Actuators:
END_STEP
TRANSITION FROM Actuators TO ActuRetract := TRUE;
END_TRANSITION
STEP ActuRetract:
	ActuRetract_action(N);
END_STEP
TRANSITION FROM ActuRetract TO ActuRetracted := checkActuator;
END_TRANSITION
STEP ActuRetracted:
	ActuRetracted_action(N);
END_STEP
STEP Lift:
END_STEP
TRANSITION FROM Lift TO StartHome := True;
END_TRANSITION
STEP StartHome:
	StartHome_action(N);
	StartHome_exit(P0);
END_STEP
TRANSITION FROM StartHome TO MoveToLoadingPos := fbDrive.bHomingDone AND tonMoveDelay.Q;
END_TRANSITION
STEP MoveToLoadingPos:
	MoveToLoadingPos_action(N);
	MoveToLoadingPos_exit(P0);
END_STEP
TRANSITION FROM MoveToLoadingPos TO DriveInLoadingPos := fbDrive.bMoveDone AND tonMoveDelay.Q;
END_TRANSITION
STEP DriveInLoadingPos:
	DriveInLoadingPos_action(N);
END_STEP
TRANSITION FROM DriveInLoadingPos TO DeliverToGarbage := bSorterLiftClear;
END_TRANSITION
STEP DeliverToGarbage:
	DeliverToGarbage_action(N);
	DeliverToGarbage_exit(P0);
END_STEP
TRANSITION FROM DeliverToGarbage TO Eject := fbDrive.bMoveDone AND tonMoveDelay.Q;
END_TRANSITION
STEP Eject:
	Eject_action(N);
	Eject_exit(P0);
END_STEP
TRANSITION FROM Eject TO ReturnToLoading := fbDelay.OK;
END_TRANSITION
STEP ReturnToLoading:
	ReturnToLoading_action(N);
	ReturnToLoading_exit(P0);
END_STEP
TRANSITION FROM ReturnToLoading TO DriveReady := fbDrive.bMoveDone AND tonMoveDelay.Q;
END_TRANSITION
STEP DriveReady:
	DriveReady_action(N);
END_STEP
TRANSITION FROM (SorterLiftClear, GatesClosed, ActuRetracted, DriveReady) TO InitMachineDone := checkAllComplete;
END_TRANSITION
STEP InitMachineDone:
	InitMachineDone_action(N);
END_STEP
TRANSITION FROM InitMachineDone TO InitMachine := NOT bExecute;
END_TRANSITION
STEP IO_Update:
END_STEP
TRANSITION FROM IO_Update TO IO_Update := TRUE;
END_TRANSITION
STEP ResetSFC:
	ResetSFC_action(N);
END_STEP
TRANSITION FROM ResetSFC TO Init := FALSE;
END_TRANSITION

ACTION Init_action:
(*Clear Reset SFC*)
SFCReset:= FALSE;
bDone := FALSE;
END_ACTION

ACTION InitMachine_action:
(*Do some actions...

Sulje kaikki portit ... JA tarkista Steppiä seuraavassa transitioehdossa, että kaikki portit ovat kiinni
Close all gates.... and check in following transition that ALL gates are closed*)

;
END_ACTION

ACTION StartInit_action:
bDone				:= FALSE;
bSorterLiftClear	:= FALSE;
bGatesClosed		:= FALSE;
bActuRetracted		:= FALSE;
bDriveAtLoading		:= FALSE;
END_ACTION

ACTION ClearAnyStuckBalls_action:
OSorterGate	:= TRUE;
tonBallClearing(IN:= TRUE, PT:= T_CLEARING_BALL , Q=> , ET=> );
END_ACTION

ACTION ClearAnyStuckBalls_exit:
tonBallClearing(IN:= FALSE);
OSorterGate	:= FALSE;
END_ACTION

ACTION SorterLiftClear_action:
bSorterLiftClear := TRUE;
END_ACTION

ACTION CloseGates_action:
OGateUp		:= FALSE;
OGateMid	:= FALSE;
OGateLow	:= FALSE;
END_ACTION

ACTION GatesClosed_action:
bGatesClosed := TRUE;
END_ACTION

ACTION ActuRetract_action:
OSorterLift	 := FALSE;
OEjector	 := FALSE;
END_ACTION

ACTION ActuRetracted_action:
bActuRetracted := TRUE;
END_ACTION

ACTION StartHome_action:
fbDrive(
	bEnable:= TRUE,
	bStart:= TRUE);

tonMoveDelay(IN:=TRUE , PT:= T_DRIVE_DELAY);
END_ACTION

ACTION StartHome_exit:
fbDrive(
	bStart:= FALSE);
END_ACTION

ACTION MoveToLoadingPos_action:
fbDrive(
	bEnable:= TRUE,
	bStart:= TRUE,
	wTarget:= GPOS_LOADING);

tonMoveDelay(IN:=TRUE , PT:= T_DRIVE_DELAY);
END_ACTION

ACTION MoveToLoadingPos_exit:
fbDrive(bStart := FALSE);
END_ACTION

ACTION DriveInLoadingPos_action:
bDriveAtLoading := TRUE;
END_ACTION

ACTION DeliverToGarbage_action:
fbDrive(
	bEnable:= TRUE,
	bStart:= TRUE,
	wTarget:= GPOS_GARBAGE);

tonMoveDelay(IN:=TRUE , PT:= T_DRIVE_DELAY);
END_ACTION

ACTION DeliverToGarbage_exit:
fbDrive(bStart := FALSE);
END_ACTION

ACTION Eject_action:
fbDelay(IN_TIME:= T_EJECTOR_DELAY, OK=> );
OEjector	 := TRUE;
END_ACTION

ACTION Eject_exit:
OEjector	 := FALSE;
END_ACTION

ACTION ReturnToLoading_action:
fbDrive(
	bEnable:= TRUE,
	bStart:= TRUE,
	wTarget:= GPOS_LOADING);

tonMoveDelay(IN:=TRUE , PT:= T_DRIVE_DELAY);
END_ACTION

ACTION ReturnToLoading_exit:
fbDrive(bStart := FALSE);
END_ACTION

ACTION DriveReady_action:
bDriveReady := TRUE;
END_ACTION

ACTION InitMachineDone_action:
bDone := TRUE;
END_ACTION

ACTION ResetSFC_action:
(*Reset SFC*)
SFCReset:=TRUE;
END_ACTION

TRANSITION CheckGates:
_FBD_ (* Function Block Diagram *)
NETWORK 1
	AND(IGateClosedUp, IGateClosedMid, IGateClosedLow)
_END_FBD_
END_TRANSITION

TRANSITION checkActuator:
_FBD_ (* Function Block Diagram *)
NETWORK 1
	AND(ISorterLiftDown, NOT OEjector)
_END_FBD_
END_TRANSITION

TRANSITION checkAllComplete:
_FBD_ (* Function Block Diagram *)
NETWORK 1
	AND(bGatesClosed, bActuRetracted, bSorterLiftClear, bDriveReady)
_END_FBD_
END_TRANSITION
END_PROGRAM

(* POU Processes/PRG_Sorting, ST *)
(* This Program performs the automatic sorting of balls into the correct locations.
when the Operator specified batch size has been completed the system enters the 
completing and bDone is Set.  Used in User mode: Sorting
Author: Nicolas Trimborn, nicolas.trimborn@tuni.fi
Date: 	2020-03-01*)

PROGRAM PRG_Sorting
VAR_INPUT
	bExecute		: BOOL;			(* Execture Auto Sorting Program *)
	bReset			: BOOL := FALSE;(* Reset Program *)
	iBatchSize  	: INT ;			(* Batch Size to Process *)
END_VAR
VAR_OUTPUT
	bDone			: BOOL;			(*Program operations done*)
	bStopOk			: BOOL;			(*Program is OK to Stop*)
	bBatchComplete  : BOOL;			(*BatchComplete *)
END_VAR
VAR
	iBallsProcessed : INT;			(* Counter for balls Processed *)
	fbSorter		: FB_Sorter;	(* FB implementation for ball sorted lift & gate *)
	fbLift			: FB_Lift;		(* FB implementation for Lift, uses FB_DriveMovement2 *)
END_VAR
IF bReset THEN (* Reset Requested *)
	bBatchComplete := FALSE;
	bDone := FALSE;
END_IF

actUpdateIO;			(* Updates I/O and calls required function blocks every cycle*)
actCheckAllOkStop;		(* Checks if lift & Sorter are both ok to stop each cycle*)
actCountBallsProcessed;	(* Counts balls processed to determine when to stop *)

CASE fbStateModel.eState OF
	eSt_Resetting:
		(*
		IF bBatchComplete THEN
			PRG_HMI.bBtnResetCounters := TRUE;
		END_IF
		*)
		fbStateModel.bSC := TRUE;
	eSt_Stopping: (* Stopping has been requested (HMI or bRun=False *)
		fbStateModel.bStop := FALSE; (* Clear Stop Flag *)

		(* Stop the Sorter and Lift FB, keep executing unitl bStopOk *)
		fbSorter(bEnable:= FALSE, bReset := FALSE);
		fbLift(bEnable:= FALSE, bReset := FALSE);
		IF bStopOk OR NOT bInitCompleted THEN (* System OK to Stop or not initialised*)
			fbStateModel.bSC := TRUE;
		END_IF
	eSt_Execute: (* Execute automatic sorting until batch Completed *)
		IF NOT bBatchComplete THEN
			fbSorter(bEnable := TRUE, bReset := FALSE);
			fbLift(bEnable := TRUE, bReset := FALSE);
		ELSE (*Stop Sorting and trigger Completing State *)
			fbSorter(bEnable := FALSE);
			fbLift(bEnable := FALSE);
			fbStateModel.bComplete := TRUE;
		END_IF

	eSt_Completing: (* Batch Has been Completed *)
		IF bStopOK THEN (* Ensure all FB are ok to stop before entering completed state *)
			bDone := TRUE;
			fbStateModel.bSC := TRUE;
		END_IF

	eSt_Unsuspending: (* Nothing Implemented *)
		fbStateModel.bSC := TRUE;

	eSt_Suspending: (* Nothing Implemented *)
		fbStateModel.bSuspend := FALSE;
		fbStateModel.bSC := TRUE;

END_CASE
END_PROGRAM
ACTION actCheckAllOKStop:
IF fbSorter.bStopOK AND  fbLift.bStopOK THEN
	bStopOK := TRUE;
ELSE
	bStopOK := FALSE;
END_IF
END_ACTION
ACTION actCountBallsProcessed:
iBallsProcessed := CountBallsSortedWooden + CountBallsSortedMetal;
iBatchRemaining := iBatchSize - iBallsProcessed;
IF iBallsProcessed >= iBatchSize  THEN
	bBatchComplete := TRUE;
ELSE
	bBatchComplete := FALSE;
END_IF
END_ACTION
ACTION actUpdateIO:
fbSorter (
	I_SensorOpt:= ISensorOpt ,
	I_SensorInd:= ISensorInd,
	I_SorterLiftUp:= ISorterLiftUp ,
	I_SorterLiftDown:= ISorterLiftDown,
	I_SorterGateClosed := ISorterGateClosed,
	hiRdyToReceive_FromDS:= fbLift.hoReadyToRecieve_ToUS ,
	hiBallAvail_FromUS:= ,
	bStopOK=> ,
	bBallLoaded=> ,
	bCurBallMetal=> ,
	O_SorterGate=> OSorterGate ,
	O_SorterLift=> OSorterLift ,
	hoBallAvail_ToDS=> ,
	hoReadyToRecieve_ToUS=> );

fbLift (
	I_LimitUp:= ILimitUp  ,
	I_LimitLow:= ILimitLow,
	I_WaitingBallMetal:= fbSorter.bCurBallMetal  ,
	I_SenColourYellow:= ISenColourYellow ,
	I_SenColourBlue:= ISenColourBlue ,
	I_SenColourGreen:= ISenColourGreen,
	I_SenColourRed:= ISenColourRed ,
	hiRdyToReceive_FromDS:= ,
	hiBallAvail_FromUS:= fbSorter.hoBallAvail_ToDS ,
	bStopOK=> ,
	bBallLoaded=> , 
	bCurBallMetal=> ,
	O_Ejector=> OEjector ,
	hoBallAvail_ToDS=> ,
	hoReadyToRecieve_ToUS=> );

(*
fbPipeUp(
	bReset:= ,
	bEnable:= bExecute,
	I_GateClosed:= IGateClosedUp ,
	I_arrCountBallsIndex:= 3,
	hiRdyToReceive_FromDS:= FALSE ,
	hiBallAvail_FromUS:= ,
	bStopOK=> ,
	bBallLoaded=> ,
	bCurBallMetal=> ,
	O_Gate=> OGateUp,
	hoBallAvail_ToDS=> FALSE ,
	hoReadyToRecieve_ToUS=> );

fbPipeMid(
	bReset:= ,
	bEnable:= bExecute,
	I_GateClosed:= IGateClosedMid,
	I_arrCountBallsIndex:= 2,
	hiRdyToReceive_FromDS:= FALSE ,
	hiBallAvail_FromUS:= ,
	bStopOK=> ,
	bBallLoaded=> ,
	bCurBallMetal=> ,
	O_Gate=> OGateMid,
	hoBallAvail_ToDS=> FALSE,
	hoReadyToRecieve_ToUS=> );

fbPipeLow(
	bReset:= ,
	bEnable:= bExecute,
	I_GateClosed:= IGateClosedLow,
	I_arrCountBallsIndex:= 1,
	hiRdyToReceive_FromDS:= FALSE,
	hiBallAvail_FromUS:= ,
	bStopOK=> ,
	bBallLoaded=> ,
	bCurBallMetal=> ,
	O_Gate=> OGateLow,
	hoBallAvail_ToDS=> FALSE,
	hoReadyToRecieve_ToUS=> );
*)
END_ACTION

(* POU FBs/FB_Sorter, SFC *)
(* This FB implements the Functionality for the SorterLift and lifts balls to the inductive
sensor based on optical sensor detecting the a ball. Handshakes are used between the lift
and sorter lifter mechanism to ensure balls arrive as expected and are delivered to the waiting
lift.

Author: Nicolas Trimborn, nicolas.trimborn@tuni.fi
Date: 	2020-03-01*)

FUNCTION_BLOCK FB_Sorter
VAR_INPUT
	bReset				: BOOL;	(*Reset Request*)
	bEnable				: BOOL;	(*Enables SorterLift*)
	I_SensorOpt			: BOOL;	(*Optical Sensor Input *)
	I_SensorInd			: BOOL;	(*Inductive Sensor Input *)
	I_SorterLiftUp		: BOOL;	(*Lift Up Sensor Input *)
	I_SorterLiftDown	: BOOL;	(*Lift Down Sensor Input *)
	I_SorterGateClosed  : BOOL;	(*Gate Closed Sensor Input *)

	(*SMEMA Handshake Inputs*)
	hiRdyToReceive_FromDS	: BOOL;
	hiBallAvail_FromUS		: BOOL;
END_VAR
VAR_OUTPUT
	O_SorterGate		: BOOL; (* Pysical output to SorterLift Gate mechanism *)
	O_SorterLift		: BOOL;	(* Pysical output to SorterLift mechanism *)

	bStopOK				: BOOL; (* FB ok to stop, not currently processing anything *)
	(* Process Flags *)
	bBallLoaded			: BOOL;
	bCurBallMetal		: BOOL;	(* Output indicating current ball is Metal or Wood *)

	(*SMEMA Handshake Outputs*)
	hoBallAvail_ToDS		: BOOL;
	hoReadyToRecieve_ToUS	: BOOL;
END_VAR
VAR
	fbInductiveTrig		: F_TRIG := (M:=FALSE); (* Falling edge trigger used to detect Metal balls rolling over sensor *)
	fbDelay				: FB_Wait;	(* Delay to allow for physical movements *)

	bLocalReset			: BOOL;	(*Performs local reset*)
	SFCReset 			: BOOL;	(*Resets the execution of SFC to init once this SFCFlag is set true *)
END_VAR
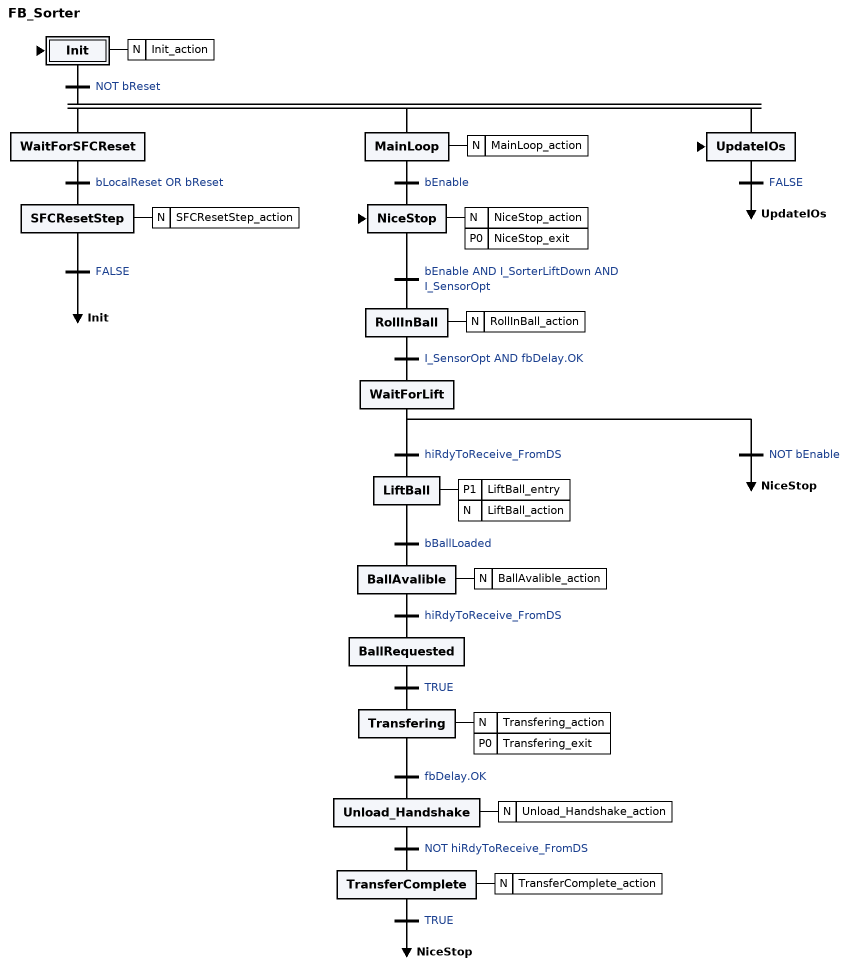
INITIAL_STEP Init:
	Init_action(N);
END_STEP
TRANSITION FROM Init TO (WaitForSFCReset, MainLoop, UpdateIOs) := NOT bReset;
END_TRANSITION
STEP WaitForSFCReset:
END_STEP
TRANSITION FROM WaitForSFCReset TO SFCResetStep := bLocalReset OR bReset;
END_TRANSITION
STEP MainLoop:
	MainLoop_action(N);
END_STEP
TRANSITION FROM MainLoop TO NiceStop := bEnable;
END_TRANSITION
STEP NiceStop:
	NiceStop_action(N);
	NiceStop_exit(P0);
END_STEP
TRANSITION FROM NiceStop TO RollInBall := bEnable AND I_SorterLiftDown AND I_SensorOpt;
END_TRANSITION
STEP RollInBall:
	RollInBall_action(N);
END_STEP
TRANSITION FROM RollInBall TO WaitForLift := I_SensorOpt AND fbDelay.OK;
END_TRANSITION
STEP WaitForLift:
END_STEP
TRANSITION FROM WaitForLift TO LiftBall := hiRdyToReceive_FromDS;
END_TRANSITION
TRANSITION FROM WaitForLift TO NiceStop := NOT bEnable;
END_TRANSITION
STEP LiftBall:
	LiftBall_entry(P1);
	LiftBall_action(N);
END_STEP
TRANSITION FROM LiftBall TO BallAvalible := bBallLoaded;
END_TRANSITION
STEP BallAvalible:
	BallAvalible_action(N);
END_STEP
TRANSITION FROM BallAvalible TO BallRequested := hiRdyToReceive_FromDS;
END_TRANSITION
STEP BallRequested:
END_STEP
TRANSITION FROM BallRequested TO Transfering := TRUE;
END_TRANSITION
STEP Transfering:
	Transfering_action(N);
	Transfering_exit(P0);
END_STEP
TRANSITION FROM Transfering TO Unload_Handshake := fbDelay.OK;
END_TRANSITION
STEP Unload_Handshake:
	Unload_Handshake_action(N);
END_STEP
TRANSITION FROM Unload_Handshake TO TransferComplete := NOT hiRdyToReceive_FromDS;
END_TRANSITION
STEP TransferComplete:
	TransferComplete_action(N);
END_STEP
TRANSITION FROM TransferComplete TO NiceStop := TRUE;
END_TRANSITION
STEP UpdateIOs:
END_STEP
TRANSITION FROM UpdateIOs TO UpdateIOs := FALSE;
END_TRANSITION
STEP SFCResetStep:
	SFCResetStep_action(N);
END_STEP
TRANSITION FROM SFCResetStep TO Init := FALSE;
END_TRANSITION

ACTION Init_action:
SFCReset := FALSE;
bLocalReset	:= FALSE;
bStopOK := TRUE;
END_ACTION

ACTION MainLoop_action:
hoBallAvail_ToDS			  := FALSE;
hoReadyToRecieve_ToUS := FALSE;
END_ACTION

ACTION NiceStop_action:
(* Clear Process Flags *)
bBallLoaded 		  := FALSE;
bStopOK				  := TRUE;

(* Ensure Gate is closed before processing ball *)
O_SorterLift 		  := FALSE;

(*Reset Handshakes *)
hoBallAvail_ToDS	  := FALSE;
hoReadyToRecieve_ToUS := FALSE;
END_ACTION

ACTION NiceStop_exit:
bStopOK := FALSE;
END_ACTION

ACTION RollInBall_action:
(* Wait for ball and account for bouncing when reloading magazine *)
fbDelay(IN_TIME:=T_BALL_DEBOUNCE);
END_ACTION

ACTION LiftBall_entry:
(*Entered processing sequence, cannot stop *)
bStopOK := FALSE;
END_ACTION

ACTION LiftBall_action:
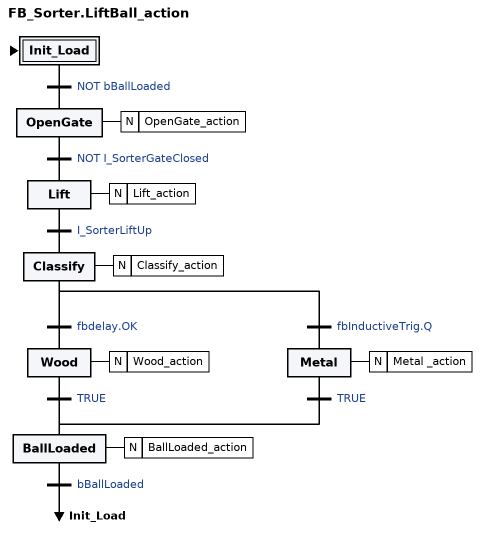
INITIAL_STEP Init_Load:
END_STEP
TRANSITION FROM Init_Load TO OpenGate := NOT bBallLoaded;
END_TRANSITION
STEP OpenGate:
	OpenGate_action(N);
END_STEP
TRANSITION FROM OpenGate TO Lift := NOT I_SorterGateClosed;
END_TRANSITION
STEP Lift:
	Lift_action(N);
END_STEP
TRANSITION FROM Lift TO Classify := I_SorterLiftUp;
END_TRANSITION
STEP Classify:
	Classify_action(N);
END_STEP
TRANSITION FROM Classify TO Wood := fbdelay.OK;
END_TRANSITION
TRANSITION FROM Classify TO Metal  := fbInductiveTrig.Q;
END_TRANSITION
STEP Wood:
	Wood_action(N);
END_STEP
TRANSITION FROM Wood TO BallLoaded := TRUE;
END_TRANSITION
STEP Metal :
	Metal _action(N);
END_STEP
TRANSITION FROM Metal  TO BallLoaded := TRUE;
END_TRANSITION
STEP BallLoaded:
	BallLoaded_action(N);
END_STEP
TRANSITION FROM BallLoaded TO Init_Load := bBallLoaded;
END_TRANSITION

ACTION OpenGate_action:
O_SorterGate := TRUE;
END_ACTION

ACTION Lift_action:
O_SorterLift := TRUE;
END_ACTION

ACTION Classify_action:
(* Wait for inductive sensor to trigger if metal ball rolls over *)
fbDelay(IN_TIME:=T_ROLL_FROM_IND);
fbInductiveTrig(CLK:=I_SensorInd);
END_ACTION

ACTION Wood_action:
bCurBallMetal := FALSE;
END_ACTION

ACTION Metal _action:
bCurBallMetal := TRUE;
END_ACTION

ACTION BallLoaded_action:
bBallLoaded := TRUE;
END_ACTION
END_ACTION

ACTION BallAvalible_action:
(*Notify Lift, ball is ready to lift *)
hoBallAvail_ToDS := TRUE;
END_ACTION

ACTION Transfering_action:
fbDelay(IN_TIME:=T_LOADING_BALL);
END_ACTION

ACTION Transfering_exit:
O_SorterGate := FALSE;
END_ACTION

ACTION Unload_Handshake_action:
(*Notify DS that ball has left SorterLift Control *)
hoBallAvail_ToDS := FALSE;
END_ACTION

ACTION TransferComplete_action:
bBallLoaded := FALSE;
END_ACTION

ACTION SFCResetStep_action:
SFCReset := TRUE;
END_ACTION
END_FUNCTION_BLOCK

(* POU FBs/FB_Lift, SFC *)
(* This FB implements the Functionality for the lifting mechanism and uses FB_DriveMovement2
provided to communicate with the drive using the Status/Control words.  Handshakes are used
between the lift and sorter lifter mechanism to ensure balls arrive as expected and are 
delivered to the appropriate tubes or colour sensor for classification

Author: Nicolas Trimborn, nicolas.trimborn@tuni.fi
Date: 	2020-03-01*)

FUNCTION_BLOCK FB_Lift
VAR_INPUT
	bReset			 	: BOOL;	(*Reset Request*)
	bEnable			 	: BOOL;	(*Enables lift*)
	I_LimitUp 			: BOOL;	(*Physical Limit switch inputs *)
	I_LimitLow 	        : BOOL;	(*Physical Limit switch inputs *)
	I_WaitingBallMetal 	: BOOL;	(*Input linked with sorter mechanism, True = Metal*)

	(* ColourSensor Inputs*)
	I_SenColourYellow	: BOOL;	(*Colour sensor In1 - Yellow*)
	I_SenColourBlue		: BOOL;	(*Colour sensor In2 - Blue*)
	I_SenColourGreen	: BOOL;	(*Colour sensor In3 - Green*)
	I_SenColourRed		: BOOL;	(*Colour sensor In4 - Red*)

	(*SMEMA Handshake Inputs*)
	hiRdyToReceive_FromDS	: BOOL;
	hiBallAvail_FromUS		: BOOL;
END_VAR
VAR_OUTPUT
	O_Ejector			: BOOL;	(* Pysical output to ejector mechanism *)

	bStopOK				: BOOL;	(* Flag set when no balls are currently being processed *)
	bBallLoaded			: BOOL;	(* Lift has a ball for processing *)
	bCurBallMetal		: BOOL;	(* Current Ball is Metal *)
	bCurrentBall 		: E_BallColour := NoColour; (*Colour of ball, NoColour is default before visiting colour sensor*)

	(*SMEMA Handshake Outputs*)
	hoBallAvail_ToDS 		: BOOL;
	hoReadyToRecieve_ToUS	: BOOL;
END_VAR
VAR
	bBallRequested 		: BOOL := FALSE; (*Flag used during material transfer from sorter lift *)

	fbDelay				: FB_Wait;	(* Delay FB used for sequencing *)
	tonSensorDelay		: TON;	(* Timer used to give time for colour sensor to perform reading*)

	bLocalReset			: BOOL;	(*Performs local reset*)
	SFCReset 			: BOOL;	(*Resets the execution of SFC to init once this SFCFlag is set true *)
END_VAR
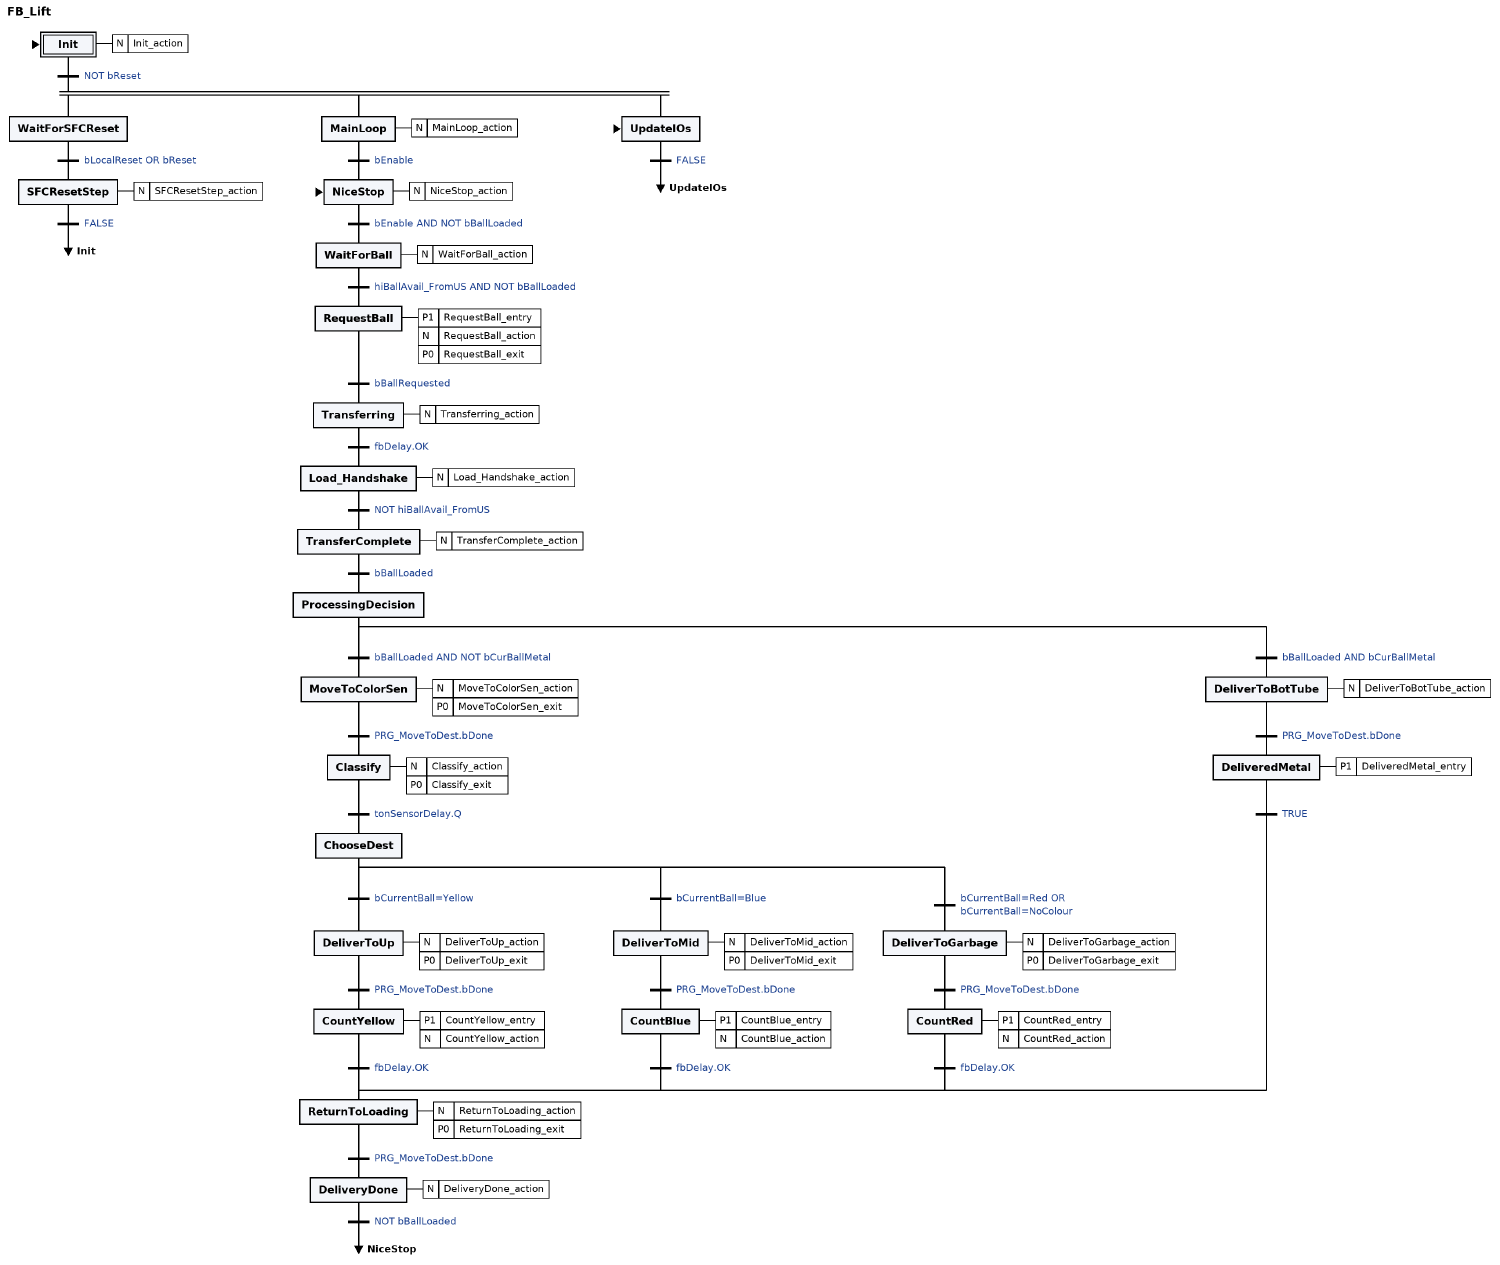
INITIAL_STEP Init:
	Init_action(N);
END_STEP
TRANSITION FROM Init TO (WaitForSFCReset, MainLoop, UpdateIOs) := NOT bReset;
END_TRANSITION
STEP WaitForSFCReset:
END_STEP
TRANSITION FROM WaitForSFCReset TO SFCResetStep := bLocalReset OR bReset;
END_TRANSITION
STEP MainLoop:
	MainLoop_action(N);
END_STEP
TRANSITION FROM MainLoop TO NiceStop := bEnable;
END_TRANSITION
STEP NiceStop:
	NiceStop_action(N);
END_STEP
TRANSITION FROM NiceStop TO WaitForBall := bEnable AND NOT bBallLoaded;
END_TRANSITION
STEP WaitForBall:
	WaitForBall_action(N);
END_STEP
TRANSITION FROM WaitForBall TO RequestBall := hiBallAvail_FromUS AND NOT bBallLoaded;
END_TRANSITION
STEP RequestBall:
	RequestBall_entry(P1);
	RequestBall_action(N);
	RequestBall_exit(P0);
END_STEP
TRANSITION FROM RequestBall TO Transferring := bBallRequested;
END_TRANSITION
STEP Transferring:
	Transferring_action(N);
END_STEP
TRANSITION FROM Transferring TO Load_Handshake := fbDelay.OK;
END_TRANSITION
STEP Load_Handshake:
	Load_Handshake_action(N);
END_STEP
TRANSITION FROM Load_Handshake TO TransferComplete := NOT hiBallAvail_FromUS;
END_TRANSITION
STEP TransferComplete:
	TransferComplete_action(N);
END_STEP
TRANSITION FROM TransferComplete TO ProcessingDecision := bBallLoaded;
END_TRANSITION
STEP ProcessingDecision:
END_STEP
TRANSITION FROM ProcessingDecision TO MoveToColorSen := bBallLoaded AND NOT bCurBallMetal;
END_TRANSITION
TRANSITION FROM ProcessingDecision TO DeliverToBotTube := bBallLoaded AND bCurBallMetal;
END_TRANSITION
STEP DeliverToBotTube:
	DeliverToBotTube_action(N);
END_STEP
TRANSITION FROM DeliverToBotTube TO DeliveredMetal := PRG_MoveToDest.bDone;
END_TRANSITION
STEP DeliveredMetal:
	DeliveredMetal_entry(P1);
END_STEP
TRANSITION FROM DeliveredMetal TO ReturnToLoading := TRUE;
END_TRANSITION
STEP MoveToColorSen:
	MoveToColorSen_action(N);
	MoveToColorSen_exit(P0);
END_STEP
TRANSITION FROM MoveToColorSen TO Classify := PRG_MoveToDest.bDone;
END_TRANSITION
STEP Classify:
	Classify_action(N);
	Classify_exit(P0);
END_STEP
TRANSITION FROM Classify TO ChooseDest := tonSensorDelay.Q;
END_TRANSITION
STEP ChooseDest:
END_STEP
TRANSITION FROM ChooseDest TO DeliverToUp := bCurrentBall=Yellow;
END_TRANSITION
TRANSITION FROM ChooseDest TO DeliverToMid := bCurrentBall=Blue;
END_TRANSITION
TRANSITION FROM ChooseDest TO DeliverToGarbage := bCurrentBall=Red OR bCurrentBall=NoColour;
END_TRANSITION
STEP DeliverToUp:
	DeliverToUp_action(N);
	DeliverToUp_exit(P0);
END_STEP
TRANSITION FROM DeliverToUp TO CountYellow := PRG_MoveToDest.bDone;
END_TRANSITION
STEP CountYellow:
	CountYellow_entry(P1);
	CountYellow_action(N);
END_STEP
TRANSITION FROM CountYellow TO ReturnToLoading := fbDelay.OK;
END_TRANSITION
STEP DeliverToMid:
	DeliverToMid_action(N);
	DeliverToMid_exit(P0);
END_STEP
TRANSITION FROM DeliverToMid TO CountBlue := PRG_MoveToDest.bDone;
END_TRANSITION
STEP CountBlue:
	CountBlue_entry(P1);
	CountBlue_action(N);
END_STEP
TRANSITION FROM CountBlue TO ReturnToLoading := fbDelay.OK;
END_TRANSITION
STEP DeliverToGarbage:
	DeliverToGarbage_action(N);
	DeliverToGarbage_exit(P0);
END_STEP
TRANSITION FROM DeliverToGarbage TO CountRed := PRG_MoveToDest.bDone;
END_TRANSITION
STEP CountRed:
	CountRed_entry(P1);
	CountRed_action(N);
END_STEP
TRANSITION FROM CountRed TO ReturnToLoading := fbDelay.OK;
END_TRANSITION
STEP ReturnToLoading:
	ReturnToLoading_action(N);
	ReturnToLoading_exit(P0);
END_STEP
TRANSITION FROM ReturnToLoading TO DeliveryDone := PRG_MoveToDest.bDone;
END_TRANSITION
STEP DeliveryDone:
	DeliveryDone_action(N);
END_STEP
TRANSITION FROM DeliveryDone TO NiceStop := NOT bBallLoaded;
END_TRANSITION
STEP UpdateIOs:
END_STEP
TRANSITION FROM UpdateIOs TO UpdateIOs := FALSE;
END_TRANSITION
STEP SFCResetStep:
	SFCResetStep_action(N);
END_STEP
TRANSITION FROM SFCResetStep TO Init := FALSE;
END_TRANSITION

ACTION Init_action:
SFCReset := FALSE;
bLocalReset	:= FALSE;
(* Initially ok to Stop *)
bStopOK := TRUE;
END_ACTION

ACTION MainLoop_action:
(* initial State of SMEMA output handshake flags *)
hoBallAvail_ToDS	  := FALSE;
hoReadyToRecieve_ToUS := FALSE;
END_ACTION

ACTION NiceStop_action:
(* Stopped initial state or state when completed processing avalible ball *)
bStopOK	  		:= TRUE;
bCurrentBall	:= NoColour;
END_ACTION

ACTION WaitForBall_action:
(* Wait for ball to become avaliable, notify US ready to recieve *)
bBallLoaded			  := FALSE;
hoReadyToRecieve_ToUS := TRUE;
END_ACTION

ACTION RequestBall_entry:
(* Processing, cannot stop until completed *)
bStopOK := FALSE;
END_ACTION

ACTION RequestBall_action:
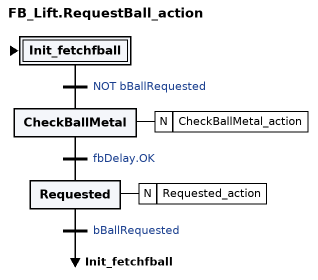
INITIAL_STEP Init_fetchfball:
END_STEP
TRANSITION FROM Init_fetchfball TO CheckBallMetal := NOT bBallRequested;
END_TRANSITION
STEP CheckBallMetal:
	CheckBallMetal_action(N);
END_STEP
TRANSITION FROM CheckBallMetal TO Requested := fbDelay.OK;
END_TRANSITION
STEP Requested:
	Requested_action(N);
END_STEP
TRANSITION FROM Requested TO Init_fetchfball := bBallRequested;
END_TRANSITION

ACTION CheckBallMetal_action:
(* Read ball type output from sorter lift,  if ball is detected as metal by IND sensor
	True = Metal
	False = Wood *)

bCurBallMetal	 := I_WaitingBallMetal;
fbDelay(IN_TIME:=T_REQ_DELAY);
END_ACTION

ACTION Requested_action:
bBallRequested := TRUE;
END_ACTION
END_ACTION

ACTION RequestBall_exit:
(* Reset Ball Requested Flag *)
bBallRequested := FALSE;
END_ACTION

ACTION Transferring_action:
(* Waiting State for ball to roll from Sorter lift to lift loading basket *)
fbDelay(IN_TIME:=T_LOADING_BALL);
END_ACTION

ACTION Load_Handshake_action:
(* Handshake to indicate ball is in control of lift *)
hoReadyToRecieve_ToUS := FALSE;
END_ACTION

ACTION TransferComplete_action:
(* When US machine no longer has a ball available, Ball transfer is complete *)
bBallLoaded := TRUE;
END_ACTION

ACTION DeliverToBotTube_action:
(* Deliver to Lower tube *)
PRG_MoveToDest(bExecute:= TRUE, wTarget:= GPOS_PIPE_LOW, bDone:= );
END_ACTION

ACTION DeliveredMetal_entry:
(* Increment Count *)
PRG_MoveToDest( bExecute:=FALSE);
CountBallsSortedMetal := CountBallsSortedMetal + 1;
arrCountBallsOnTubes[1] := arrCountBallsOnTubes[1] + 1;
END_ACTION

ACTION MoveToColorSen_action:
(* Send Wooden Ball to colour sensor for evaluation *)
PRG_MoveToDest(bExecute:= TRUE, wTarget:= GPOS_COLOR_SEN, bDone:= );
END_ACTION

ACTION MoveToColorSen_exit:
PRG_MoveToDest( bExecute:=FALSE);
END_ACTION

ACTION Classify_action:
(* Read Colour Sensor Inputs *)
tonSensorDelay(IN:=TRUE , PT:= T_COLOUR_SENSOR_DELAY);
IF I_SenColourYellow THEN
	bCurrentBall := Yellow;
ELSIF  I_SenColourBlue THEN
	bCurrentBall := Blue;
ELSIF  I_SenColourRed THEN
	bCurrentBall := Red;
ELSE (* Unclassified balls sent to garbage chute *)
	bCurrentBall := NoColour;
END_IF
END_ACTION

ACTION Classify_exit:
tonSensorDelay(IN:=FALSE);
END_ACTION

ACTION DeliverToUp_action:
PRG_MoveToDest(bExecute:= TRUE , wTarget:= GPOS_PIPE_UP, bDone:= );
END_ACTION

ACTION DeliverToUp_exit:
PRG_MoveToDest(bExecute:= FALSE);
END_ACTION

ACTION CountYellow_entry:
CountBallsSortedYellow := CountBallsSortedYellow + 1;
CountBallsSortedWooden := CountBallsSortedWooden + 1;
arrCountBallsOnTubes[3] := arrCountBallsOnTubes[3] + 1;
END_ACTION

ACTION CountYellow_action:
fbDelay(IN_TIME:=T_POS_SETTLE_DELAY);
END_ACTION

ACTION DeliverToMid_action:
PRG_MoveToDest(bExecute:= TRUE , wTarget:= GPOS_PIPE_MID, bDone:= );
END_ACTION

ACTION DeliverToMid_exit:
PRG_MoveToDest(bExecute:= FALSE);
END_ACTION

ACTION CountBlue_entry:
CountBallsSortedBlue := CountBallsSortedBlue + 1;
CountBallsSortedWooden := CountBallsSortedWooden + 1;
arrCountBallsOnTubes[2] := arrCountBallsOnTubes[2] + 1;
END_ACTION

ACTION CountBlue_action:
fbDelay(IN_TIME:=T_POS_SETTLE_DELAY);
END_ACTION

ACTION DeliverToGarbage_action:
PRG_MoveToDest(bExecute:= TRUE , wTarget:= GPOS_GARBAGE, bDone:= );
END_ACTION

ACTION DeliverToGarbage_exit:
PRG_MoveToDest(bExecute:= FALSE);
END_ACTION

ACTION CountRed_entry:
CountBallsSortedRed := CountBallsSortedRed + 1;
CountBallsSortedGarbage := CountBallsSortedGarbage + 1;
CountBallsSortedWooden := CountBallsSortedWooden + 1;
arrCountBallsOnTubes[4] := arrCountBallsOnTubes[4] + 1;
END_ACTION

ACTION CountRed_action:
fbDelay(IN_TIME:=T_POS_SETTLE_DELAY);
END_ACTION

ACTION ReturnToLoading_action:
PRG_MoveToDest(bExecute:= TRUE , wTarget:= GPOS_LOADING, bDone:= );
END_ACTION

ACTION ReturnToLoading_exit:
PRG_MoveToDest(bExecute:= FALSE);
END_ACTION

ACTION DeliveryDone_action:
(* Ball Sorting operation Completed *)
bBallLoaded := FALSE;
bCurrentBall := NoColour;
END_ACTION

ACTION SFCResetStep_action:
SFCReset := TRUE;
END_ACTION
END_FUNCTION_BLOCK

(* POU Processes/PRG_MoveToDest, SFC *)
PROGRAM PRG_MoveToDest
VAR_INPUT
	bExecute: BOOL;
	wTarget : WORD;
END_VAR
VAR_INPUT
	bDone: BOOL;
END_VAR
VAR
	tonMoveDelay	: TON;
	tonEjectDelay	: TON;
	tonSensorDelay	: TON;
	tMoveDelay		: TIME := T#500ms;
	tEjectorDelay	: TIME := T#1s;
	tSensorDelay	: TIME := T#500ms;
END_VAR
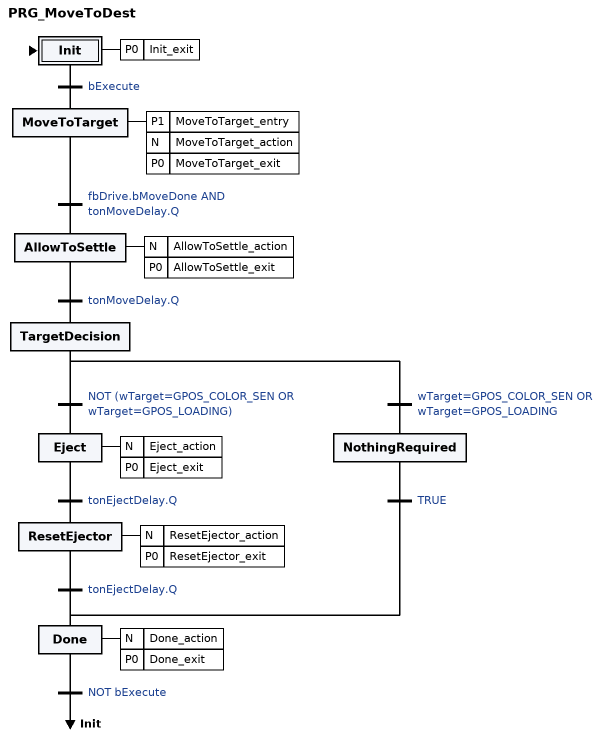
INITIAL_STEP Init:
	Init_exit(P0);
END_STEP
TRANSITION FROM Init TO MoveToTarget := bExecute;
END_TRANSITION
STEP MoveToTarget:
	MoveToTarget_entry(P1);
	MoveToTarget_action(N);
	MoveToTarget_exit(P0);
END_STEP
TRANSITION FROM MoveToTarget TO AllowToSettle := fbDrive.bMoveDone AND tonMoveDelay.Q;
END_TRANSITION
STEP AllowToSettle:
	AllowToSettle_action(N);
	AllowToSettle_exit(P0);
END_STEP
TRANSITION FROM AllowToSettle TO TargetDecision := tonMoveDelay.Q;
END_TRANSITION
STEP TargetDecision:
END_STEP
TRANSITION FROM TargetDecision TO Eject := NOT (wTarget=GPOS_COLOR_SEN OR wTarget=GPOS_LOADING);
END_TRANSITION
TRANSITION FROM TargetDecision TO NothingRequired := wTarget=GPOS_COLOR_SEN OR wTarget=GPOS_LOADING;
END_TRANSITION
STEP NothingRequired:
END_STEP
TRANSITION FROM NothingRequired TO Done := TRUE;
END_TRANSITION
STEP Eject:
	Eject_action(N);
	Eject_exit(P0);
END_STEP
TRANSITION FROM Eject TO ResetEjector := tonEjectDelay.Q;
END_TRANSITION
STEP ResetEjector:
	ResetEjector_action(N);
	ResetEjector_exit(P0);
END_STEP
TRANSITION FROM ResetEjector TO Done := tonEjectDelay.Q;
END_TRANSITION
STEP Done:
	Done_action(N);
	Done_exit(P0);
END_STEP
TRANSITION FROM Done TO Init := NOT bExecute;
END_TRANSITION

ACTION Init_exit:
bDone := FALSE;
END_ACTION

ACTION MoveToTarget_entry:
tonMoveDelay(IN:=FALSE);
fbDrive(bStart:= FALSE);
END_ACTION

ACTION MoveToTarget_action:
(*Drive Move Delay *)
tonMoveDelay(IN:=TRUE, PT:= T_DRIVE_DELAY);
(* Drive To Target *)
fbDrive(
	bEnable:= TRUE,
	bStart:= TRUE,
	wTarget:= wTarget);
END_ACTION

ACTION MoveToTarget_exit:
fbDrive(
	bStart:= FALSE);
tonMoveDelay(IN:=FALSE);
END_ACTION

ACTION AllowToSettle_action:
tonMoveDelay(IN:=TRUE , PT:= T_POS_SETTLE_DELAY);
END_ACTION

ACTION AllowToSettle_exit:
tonMoveDelay(IN:=FALSE);
END_ACTION

ACTION Eject_action:
tonEjectDelay(IN:=TRUE , PT:= T_EJECTOR_DELAY);
OEjector := TRUE;
END_ACTION

ACTION Eject_exit:
tonEjectDelay(IN:=FALSE);
END_ACTION

ACTION ResetEjector_action:
(* Retract Ejector *)
tonEjectDelay(IN:=TRUE , PT:= T_EJECTOR_DELAY);
OEjector := FALSE;
END_ACTION

ACTION ResetEjector_exit:
tonEjectDelay(IN:=FALSE);
END_ACTION

ACTION Done_action:
bDone := TRUE;
END_ACTION

ACTION Done_exit:
bDone := FALSE;
END_ACTION
END_PROGRAM

(* POU Background Programs/PRG_Drive_Link, FBD *)
PROGRAM PRG_Drive_Link
VAR
END_VAR
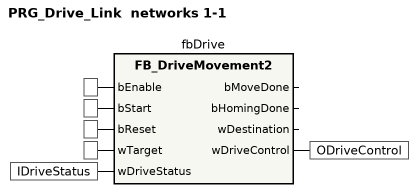
_FBD_ (* Function Block Diagram *)
NETWORK 1
	fbDrive:FB_DriveMovement2(bEnable: , bStart: , bReset: , wTarget: , wDriveStatus: IDriveStatus, wDriveControl => ODriveControl)
_END_FBD_
END_PROGRAM

(* POU FBs/FB_DriveMovement2, ST *)
FUNCTION_BLOCK FB_DriveMovement2
(* This function block is making all movements for the drive
	bEnable = must be TRUE
	Target = int value of 0 - 63
	bStart = with rising edge starts the movement

	bMoveDone gets true when the movement is finalised.
Author: 	Niko Siltala, niko.siltala@tut.fi
Date: 	2014-01-01*)

VAR_INPUT
	bEnable			: BOOL:=FALSE;	(*Enables the fuction block*)
	bStart			: BOOL:=FALSE;	(*Starts the motion to target by rising edge*)
	bReset			: BOOL:=FALSE;
	wTarget			: WORD:=0;		(*Target destination*)
	wDriveStatus		: WORD;			(*Status word from Indramat Drive*)
END_VAR
VAR_OUTPUT
	bMoveDone		:BOOL:=FALSE;	(*The commanded move has been completed. Drive is at required destination*)
	bHomingDone	:BOOL:=FALSE;	(*Drive has been homed*)
	wDestination		:WORD;			(*Current destination*)
	wDriveControl		:WORD;			(*Control word to Indramat Drive*)
END_VAR
VAR_IN_OUT
END_VAR
VAR
	TONTimer1 	: TON;
	TONTimer2 	: TON;
END_VAR
(*
This function block is making all movements for the drive
	bEnable = must be TRUE
	Target = int value of 0 - 63
	bStart = with rising edge starts the movement

	bMoveDone gets true when the movement is finalised
*)


IF bEnable THEN
	(*Drive is Enabled*)
	wDriveControl:=wDriveControl OR 16#0001;
	IF (wDriveStatus AND 16#0080)>0 AND (wDriveStatus AND 16#0040)>0 THEN
		IF bStart=TRUE THEN
			(*bStart is true*)
			IF bHomingDone=FALSE THEN
				(*Homing procedure*)
				IF TONTimer1.Q=FALSE THEN
					wDriveControl:=16#0005;
					TONTimer1(IN:=TRUE, PT:=T#100ms);(*100ms*)
				ELSE
					IF TONTimer2.Q=FALSE THEN
						(*Start drive*)
						wDriveControl:=16#0007;
						TONTimer2(IN:=TRUE, PT:=T#500ms); (*500ms*)
					ELSE
						(*Timer2 have expired*)
						IF (wDriveStatus AND 16#0004)>0 THEN
							TONTimer1(IN:=FALSE);
							TONTimer2(IN:=FALSE);
							wDriveControl:=16#0001;
							bHomingDone:=TRUE;
						END_IF;
					END_IF;
				END_IF;
			ELSE
				(*Normal movement*)
				IF TONTimer1.Q=FALSE THEN
					(*Set target and Enabled*)
					wDriveControl:=SHL(wTarget,8) OR 16#0001;
					wDestination:=wTarget;
					TONTimer1(IN:=TRUE, PT:=T#10ms);(*10ms*)
				ELSE
					IF TONTimer2.Q=FALSE THEN
						(*Start drive*)
						wDriveControl:=wDriveControl OR 16#0002;
						TONTimer2(IN:=TRUE, PT:=T#500ms); (*500ms*)
					ELSE
						(*Timer2 have expired*)
						IF (wDriveStatus AND 16#0010)>0 THEN
							(*End the movement when user forgets to provide lowering edge*)
							bStart:=FALSE;
							(*Requested movement is done*)
							bMoveDone:=TRUE;
						END_IF;
					END_IF;
				END_IF; (*Normal movement*)
			END_IF;(*bHomingDone=FALSE*)
		ELSE
			(*bStart is false*)
			bMoveDone:=FALSE;
			TONTimer1(IN:=FALSE);
			TONTimer2(IN:=FALSE);
		END_IF;
	END_IF;
	(* Reset Drive Errors by seeting FReset Bit *)
	IF bReset THEN
		wDriveControl.5 := TRUE;
	ELSE
		wDriveControl.5 := FALSE;
	END_IF;
ELSE (*bEnable*)
	(*Drive is NOT Enabled*)
	wDriveControl:=16#0000;
	bMoveDone:=FALSE;
	bHomingDone:=FALSE;
	TONTimer1(IN:=FALSE);
	TONTimer2(IN:=FALSE);
	(* Reset Drive Errors by seeting FReset Bit *)
	IF bReset THEN
		wDriveControl.5 := TRUE;
	ELSE
		wDriveControl.5 := FALSE;
	END_IF;
END_IF;
END_FUNCTION_BLOCK

(* POU PRG_SafetyProgram, ST *)
PROGRAM PRG_SafetyProgram
VAR
END_VAR
IF NOT IEmergencyClear OR ILimitLow OR ILimitUp THEN
	ODriveControl := 16#0000;
	fbDrive(bEnable:= FALSE, bStart := FALSE);
END_IF
END_PROGRAM

(* POU Example/EXAMPLES, SFC *)
PROGRAM EXAMPLES
VAR
	fbDrive			: DriveMovement2;		(*FB for executing the motion*)
	tonTimer			: TON;			(*Standard TON timer. Use this*)
	fbDelay			: FB_Wait;		(*Different simplified timer.
END_VAR
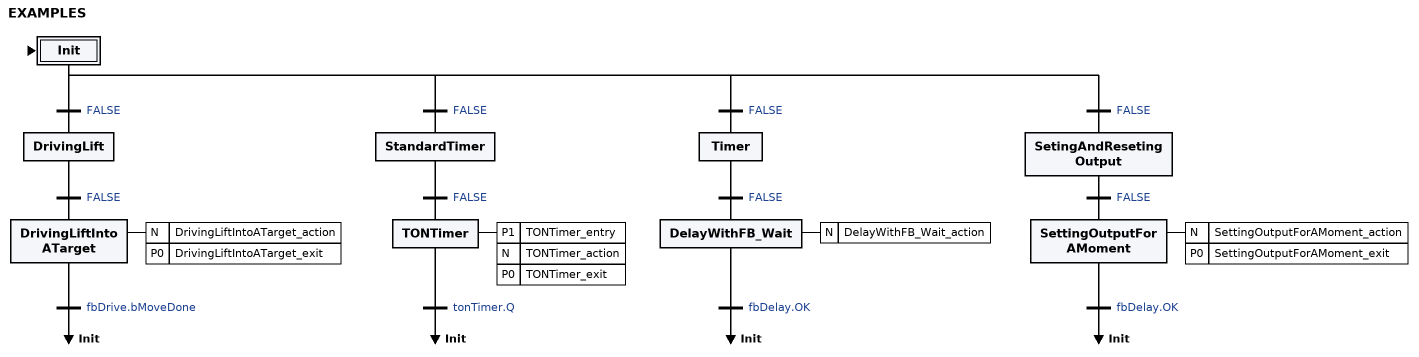
INITIAL_STEP Init:
END_STEP
TRANSITION FROM Init TO DrivingLift := FALSE;
END_TRANSITION
TRANSITION FROM Init TO StandardTimer := FALSE;
END_TRANSITION
TRANSITION FROM Init TO Timer := FALSE;
END_TRANSITION
TRANSITION FROM Init TO SetingAndResetingOutput := FALSE;
END_TRANSITION
STEP DrivingLift:
END_STEP
TRANSITION FROM DrivingLift TO DrivingLiftIntoATarget := FALSE;
END_TRANSITION
STEP DrivingLiftIntoATarget:
	DrivingLiftIntoATarget_action(N);
	DrivingLiftIntoATarget_exit(P0);
END_STEP
TRANSITION FROM DrivingLiftIntoATarget TO Init := fbDrive.bMoveDone;
END_TRANSITION
STEP StandardTimer:
END_STEP
TRANSITION FROM StandardTimer TO TONTimer := FALSE;
END_TRANSITION
STEP TONTimer:
	TONTimer_entry(P1);
	TONTimer_action(N);
	TONTimer_exit(P0);
END_STEP
TRANSITION FROM TONTimer TO Init := tonTimer.Q;
END_TRANSITION
STEP Timer:
END_STEP
TRANSITION FROM Timer TO DelayWithFB_Wait := FALSE;
END_TRANSITION
STEP DelayWithFB_Wait:
	DelayWithFB_Wait_action(N);
END_STEP
TRANSITION FROM DelayWithFB_Wait TO Init := fbDelay.OK;
END_TRANSITION
STEP SetingAndResetingOutput:
END_STEP
TRANSITION FROM SetingAndResetingOutput TO SettingOutputForAMoment := FALSE;
END_TRANSITION
STEP SettingOutputForAMoment:
	SettingOutputForAMoment_action(N);
	SettingOutputForAMoment_exit(P0);
END_STEP
TRANSITION FROM SettingOutputForAMoment TO Init := fbDelay.OK;
END_TRANSITION

ACTION DrivingLiftIntoATarget_action:
(*This executes and drives the lift to desired level (=wTarget)
wTarget is selected from given constants. See:Global Constants*)
fbDrive(
	bEnable:= TRUE,
	bStart:= TRUE,
	wTarget:= GPOS_LOADING);
END_ACTION

ACTION DrivingLiftIntoATarget_exit:
(*Stops the motion*)
fbDrive(
	bStart:= FALSE);
END_ACTION

ACTION TONTimer_entry:
tonTimer(IN:=FALSE);
END_ACTION

ACTION TONTimer_action:
tonTimer(IN:=TRUE , PT:=T#1s, Q=> , ET=> );
END_ACTION

ACTION TONTimer_exit:
tonTimer(IN:=FALSE);
END_ACTION

ACTION DelayWithFB_Wait_action:
(*Timer is counting*)
fbDelay(IN_TIME:=T#1s);
END_ACTION

ACTION SettingOutputForAMoment_action:
(*Timer is counting*)
fbDelay(IN_TIME:=T#500ms);

(*Setting Output*)
OEjector := TRUE;
END_ACTION

ACTION SettingOutputForAMoment_exit:
(*Clearing Output*)
OEjector := FALSE;
END_ACTION
END_PROGRAM

(* POU OLD/PRG_DeliverToGarbage, SFC *)
PROGRAM PRG_DeliverToGarbage
VAR_INPUT
	bReset		: BOOL;	(*Reset program*)
	bExecute		: BOOL;	(*enable and run*)
END_VAR
VAR_OUTPUT
	bDone			: BOOL;
END_VAR
VAR
	tonMoveDelay	: TON;
	tonEjectDelay	: TON;
	SFCReset		: BOOL;

	tMoveDelay	: TIME := T#4s;
	tEjectorDelay	: TIME := T#2s;
END_VAR
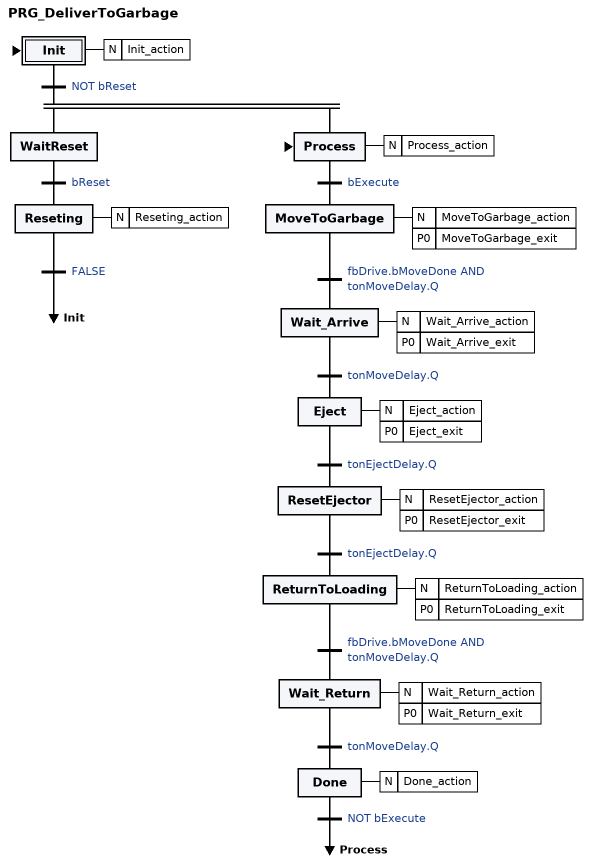
INITIAL_STEP Init:
	Init_action(N);
END_STEP
TRANSITION FROM Init TO (WaitReset, Process) := NOT bReset;
END_TRANSITION
STEP WaitReset:
END_STEP
TRANSITION FROM WaitReset TO Reseting := bReset;
END_TRANSITION
STEP Process:
	Process_action(N);
END_STEP
TRANSITION FROM Process TO MoveToGarbage := bExecute;
END_TRANSITION
STEP MoveToGarbage:
	MoveToGarbage_action(N);
	MoveToGarbage_exit(P0);
END_STEP
TRANSITION FROM MoveToGarbage TO Wait_Arrive := fbDrive.bMoveDone AND tonMoveDelay.Q;
END_TRANSITION
STEP Wait_Arrive:
	Wait_Arrive_action(N);
	Wait_Arrive_exit(P0);
END_STEP
TRANSITION FROM Wait_Arrive TO Eject := tonMoveDelay.Q;
END_TRANSITION
STEP Eject:
	Eject_action(N);
	Eject_exit(P0);
END_STEP
TRANSITION FROM Eject TO ResetEjector := tonEjectDelay.Q;
END_TRANSITION
STEP ResetEjector:
	ResetEjector_action(N);
	ResetEjector_exit(P0);
END_STEP
TRANSITION FROM ResetEjector TO ReturnToLoading := tonEjectDelay.Q;
END_TRANSITION
STEP ReturnToLoading:
	ReturnToLoading_action(N);
	ReturnToLoading_exit(P0);
END_STEP
TRANSITION FROM ReturnToLoading TO Wait_Return := fbDrive.bMoveDone AND tonMoveDelay.Q;
END_TRANSITION
STEP Wait_Return:
	Wait_Return_action(N);
	Wait_Return_exit(P0);
END_STEP
TRANSITION FROM Wait_Return TO Done := tonMoveDelay.Q;
END_TRANSITION
STEP Done:
	Done_action(N);
END_STEP
TRANSITION FROM Done TO Process := NOT bExecute;
END_TRANSITION
STEP Reseting:
	Reseting_action(N);
END_STEP
TRANSITION FROM Reseting TO Init := FALSE;
END_TRANSITION

ACTION Init_action:
SFCReset := FALSE;
bDone := FALSE;
END_ACTION

ACTION Process_action:
bDone := FALSE;
END_ACTION

ACTION MoveToGarbage_action:
bDone := FALSE;

fbDrive(
	bEnable:= TRUE,
	bStart:= TRUE,
	wTarget:= GPOS_GARBAGE);

tonMoveDelay(IN:=TRUE , PT:= tMoveDelay);
END_ACTION

ACTION MoveToGarbage_exit:
fbDrive(
	bStart:= FALSE);

tonMoveDelay(IN:=FALSE);
END_ACTION

ACTION Wait_Arrive_action:
tonMoveDelay(IN:=TRUE , PT:= tMoveDelay);
END_ACTION

ACTION Wait_Arrive_exit:
tonMoveDelay(IN:=FALSE);
END_ACTION

ACTION Eject_action:
OEjector := TRUE;
tonEjectDelay(IN:=TRUE , PT:= tEjectorDelay);
END_ACTION

ACTION Eject_exit:
tonEjectDelay(IN:=FALSE);
END_ACTION

ACTION ResetEjector_action:
OEjector := FALSE;
tonEjectDelay(IN:=TRUE , PT:= tEjectorDelay);
END_ACTION

ACTION ResetEjector_exit:
tonEjectDelay(IN:=FALSE);
END_ACTION

ACTION ReturnToLoading_action:
fbDrive(
	bEnable:= TRUE,
	bStart:= TRUE,
	wTarget:= GPOS_LOADING);

tonMoveDelay(IN:=TRUE , PT:= tMoveDelay);
END_ACTION

ACTION ReturnToLoading_exit:
fbDrive(
	bStart:= FALSE);

tonMoveDelay(IN:=FALSE);
END_ACTION

ACTION Wait_Return_action:
tonMoveDelay(IN:=TRUE , PT:= tMoveDelay);
END_ACTION

ACTION Wait_Return_exit:
tonMoveDelay(IN:=FALSE);
END_ACTION

ACTION Done_action:
bDone := TRUE;
END_ACTION

ACTION Reseting_action:
SFCReset := TRUE;
END_ACTION
END_PROGRAM

(* POU OLD/PRG_DeliverToGarbage2, SFC *)
PROGRAM PRG_DeliverToGarbage2
VAR_INPUT
	bExecute: BOOL;
END_VAR
VAR_INPUT
	bDone: BOOL;
END_VAR
VAR
	tonMoveDelay	: TON;
	tonEjectDelay	: TON;
	tMoveDelay	: TIME := T#3s;
	tEjectorDelay	: TIME := T#3s;
END_VAR
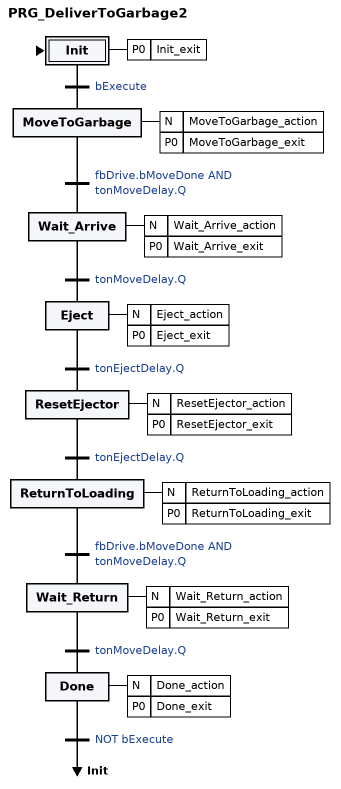
INITIAL_STEP Init:
	Init_exit(P0);
END_STEP
TRANSITION FROM Init TO MoveToGarbage := bExecute;
END_TRANSITION
STEP MoveToGarbage:
	MoveToGarbage_action(N);
	MoveToGarbage_exit(P0);
END_STEP
TRANSITION FROM MoveToGarbage TO Wait_Arrive := fbDrive.bMoveDone AND tonMoveDelay.Q;
END_TRANSITION
STEP Wait_Arrive:
	Wait_Arrive_action(N);
	Wait_Arrive_exit(P0);
END_STEP
TRANSITION FROM Wait_Arrive TO Eject := tonMoveDelay.Q;
END_TRANSITION
STEP Eject:
	Eject_action(N);
	Eject_exit(P0);
END_STEP
TRANSITION FROM Eject TO ResetEjector := tonEjectDelay.Q;
END_TRANSITION
STEP ResetEjector:
	ResetEjector_action(N);
	ResetEjector_exit(P0);
END_STEP
TRANSITION FROM ResetEjector TO ReturnToLoading := tonEjectDelay.Q;
END_TRANSITION
STEP ReturnToLoading:
	ReturnToLoading_action(N);
	ReturnToLoading_exit(P0);
END_STEP
TRANSITION FROM ReturnToLoading TO Wait_Return := fbDrive.bMoveDone AND tonMoveDelay.Q;
END_TRANSITION
STEP Wait_Return:
	Wait_Return_action(N);
	Wait_Return_exit(P0);
END_STEP
TRANSITION FROM Wait_Return TO Done := tonMoveDelay.Q;
END_TRANSITION
STEP Done:
	Done_action(N);
	Done_exit(P0);
END_STEP
TRANSITION FROM Done TO Init := NOT bExecute;
END_TRANSITION

ACTION Init_exit:
bDone := FALSE;
END_ACTION

ACTION MoveToGarbage_action:
fbDrive(
	bEnable:= TRUE,
	bStart:= TRUE,
	wTarget:= GPOS_GARBAGE);

tonMoveDelay(IN:=TRUE , PT:= tMoveDelay);
END_ACTION

ACTION MoveToGarbage_exit:
fbDrive(
	bStart:= FALSE);
tonMoveDelay(IN:=FALSE);
END_ACTION

ACTION Wait_Arrive_action:
tonMoveDelay(IN:=TRUE , PT:= tMoveDelay);
END_ACTION

ACTION Wait_Arrive_exit:
tonMoveDelay(IN:=FALSE);
END_ACTION

ACTION Eject_action:
OEjector := TRUE;
tonEjectDelay(IN:=TRUE , PT:= tEjectorDelay);
END_ACTION

ACTION Eject_exit:
tonEjectDelay(IN:=FALSE);
END_ACTION

ACTION ResetEjector_action:
OEjector := FALSE;
tonEjectDelay(IN:=TRUE , PT:= tEjectorDelay);
END_ACTION

ACTION ResetEjector_exit:
tonEjectDelay(IN:=FALSE);
END_ACTION

ACTION ReturnToLoading_action:
fbDrive(
	bEnable:= TRUE,
	bStart:= TRUE,
	wTarget:= GPOS_LOADING);

tonMoveDelay(IN:=TRUE , PT:= tMoveDelay);
END_ACTION

ACTION ReturnToLoading_exit:
fbDrive(
	bStart:= FALSE);

tonMoveDelay(IN:=FALSE);
END_ACTION

ACTION Wait_Return_action:
tonMoveDelay(IN:=TRUE , PT:= tMoveDelay);
END_ACTION

ACTION Wait_Return_exit:
tonMoveDelay(IN:=FALSE);
END_ACTION

ACTION Done_action:
bDone := TRUE;
END_ACTION

ACTION Done_exit:
bDone := FALSE;
END_ACTION
END_PROGRAM

(* POU OLD/PRG_DeliverToLow, SFC *)
PROGRAM PRG_DeliverToLow
VAR_INPUT
	bReset		: BOOL;	(*Reset program*)
	bExecute		: BOOL;	(*enable and run*)

END_VAR
VAR_OUTPUT
	bDone			: BOOL;
END_VAR
VAR
	tonMoveDelay	: TON;
	tonEjectDelay	: TON;
	SFCReset		: BOOL;

	tMoveDelay	: TIME := T#4s;
	tEjectorDelay	: TIME := T#3s;
END_VAR
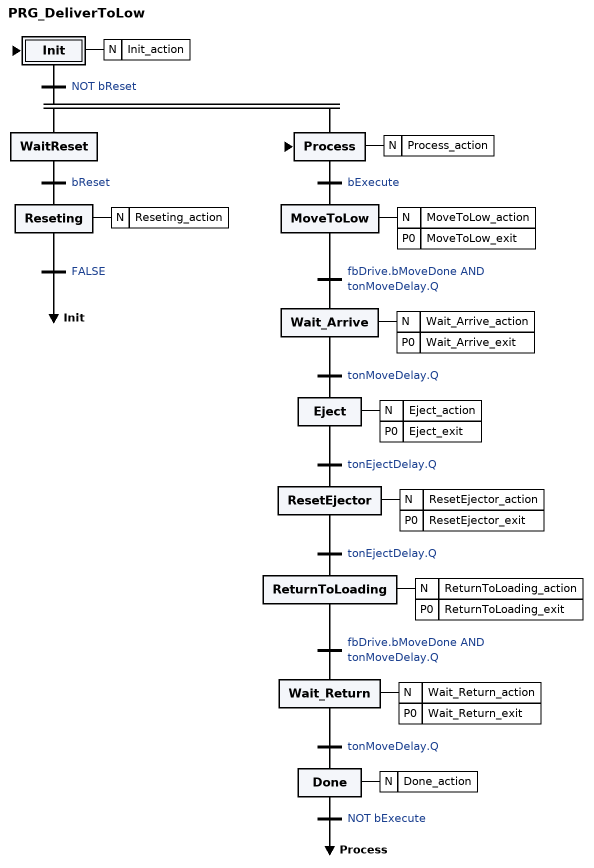
INITIAL_STEP Init:
	Init_action(N);
END_STEP
TRANSITION FROM Init TO (WaitReset, Process) := NOT bReset;
END_TRANSITION
STEP WaitReset:
END_STEP
TRANSITION FROM WaitReset TO Reseting := bReset;
END_TRANSITION
STEP Process:
	Process_action(N);
END_STEP
TRANSITION FROM Process TO MoveToLow := bExecute;
END_TRANSITION
STEP MoveToLow:
	MoveToLow_action(N);
	MoveToLow_exit(P0);
END_STEP
TRANSITION FROM MoveToLow TO Wait_Arrive := fbDrive.bMoveDone AND tonMoveDelay.Q;
END_TRANSITION
STEP Wait_Arrive:
	Wait_Arrive_action(N);
	Wait_Arrive_exit(P0);
END_STEP
TRANSITION FROM Wait_Arrive TO Eject := tonMoveDelay.Q;
END_TRANSITION
STEP Eject:
	Eject_action(N);
	Eject_exit(P0);
END_STEP
TRANSITION FROM Eject TO ResetEjector := tonEjectDelay.Q;
END_TRANSITION
STEP ResetEjector:
	ResetEjector_action(N);
	ResetEjector_exit(P0);
END_STEP
TRANSITION FROM ResetEjector TO ReturnToLoading := tonEjectDelay.Q;
END_TRANSITION
STEP ReturnToLoading:
	ReturnToLoading_action(N);
	ReturnToLoading_exit(P0);
END_STEP
TRANSITION FROM ReturnToLoading TO Wait_Return := fbDrive.bMoveDone AND tonMoveDelay.Q;
END_TRANSITION
STEP Wait_Return:
	Wait_Return_action(N);
	Wait_Return_exit(P0);
END_STEP
TRANSITION FROM Wait_Return TO Done := tonMoveDelay.Q;
END_TRANSITION
STEP Done:
	Done_action(N);
END_STEP
TRANSITION FROM Done TO Process := NOT bExecute;
END_TRANSITION
STEP Reseting:
	Reseting_action(N);
END_STEP
TRANSITION FROM Reseting TO Init := FALSE;
END_TRANSITION

ACTION Init_action:
SFCReset := FALSE;
bDone := FALSE;
END_ACTION

ACTION Process_action:
bDone := FALSE;
END_ACTION

ACTION MoveToLow_action:
bDone := FALSE;

fbDrive(
	bEnable:= TRUE,
	bStart:= TRUE,
	wTarget:= GPOS_PIPE_LOW);

tonMoveDelay(IN:=TRUE , PT:= tMoveDelay);
END_ACTION

ACTION MoveToLow_exit:
fbDrive(
	bStart:= FALSE);
tonMoveDelay(IN:=FALSE);
END_ACTION

ACTION Wait_Arrive_action:
tonMoveDelay(IN:=TRUE , PT:= tMoveDelay);
END_ACTION

ACTION Wait_Arrive_exit:
tonMoveDelay(IN:=FALSE);
END_ACTION

ACTION Eject_action:
OEjector := TRUE;
tonEjectDelay(IN:=TRUE , PT:= tEjectorDelay);
END_ACTION

ACTION Eject_exit:
tonEjectDelay(IN:=FALSE);
END_ACTION

ACTION ResetEjector_action:
OEjector := FALSE;
tonEjectDelay(IN:=TRUE , PT:= tEjectorDelay);
END_ACTION

ACTION ResetEjector_exit:
tonEjectDelay(IN:=FALSE);
END_ACTION

ACTION ReturnToLoading_action:
fbDrive(
	bEnable:= TRUE,
	bStart:= TRUE,
	wTarget:= GPOS_LOADING);

tonMoveDelay(IN:=TRUE , PT:= tMoveDelay);
END_ACTION

ACTION ReturnToLoading_exit:
fbDrive(
	bStart:= FALSE);

tonMoveDelay(IN:=FALSE);
END_ACTION

ACTION Wait_Return_action:
tonMoveDelay(IN:=TRUE , PT:= tMoveDelay);
END_ACTION

ACTION Wait_Return_exit:
tonMoveDelay(IN:=FALSE);
END_ACTION

ACTION Done_action:
bDone := TRUE;
END_ACTION

ACTION Reseting_action:
SFCReset := TRUE;
END_ACTION
END_PROGRAM

(* POU OLD/PRG_DeliverToLow2, SFC *)
PROGRAM PRG_DeliverToLow2
VAR_INPUT
	bExecute: BOOL;
END_VAR
VAR_INPUT
	bDone: BOOL;
END_VAR
VAR
	tonMoveDelay	: TON;
	tonEjectDelay	: TON;
	tMoveDelay	: TIME := T#4s;
	tEjectorDelay	: TIME := T#3s;
END_VAR
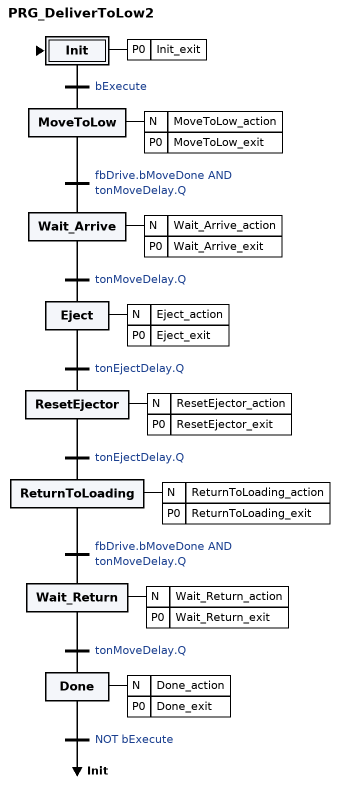
INITIAL_STEP Init:
	Init_exit(P0);
END_STEP
TRANSITION FROM Init TO MoveToLow := bExecute;
END_TRANSITION
STEP MoveToLow:
	MoveToLow_action(N);
	MoveToLow_exit(P0);
END_STEP
TRANSITION FROM MoveToLow TO Wait_Arrive := fbDrive.bMoveDone AND tonMoveDelay.Q;
END_TRANSITION
STEP Wait_Arrive:
	Wait_Arrive_action(N);
	Wait_Arrive_exit(P0);
END_STEP
TRANSITION FROM Wait_Arrive TO Eject := tonMoveDelay.Q;
END_TRANSITION
STEP Eject:
	Eject_action(N);
	Eject_exit(P0);
END_STEP
TRANSITION FROM Eject TO ResetEjector := tonEjectDelay.Q;
END_TRANSITION
STEP ResetEjector:
	ResetEjector_action(N);
	ResetEjector_exit(P0);
END_STEP
TRANSITION FROM ResetEjector TO ReturnToLoading := tonEjectDelay.Q;
END_TRANSITION
STEP ReturnToLoading:
	ReturnToLoading_action(N);
	ReturnToLoading_exit(P0);
END_STEP
TRANSITION FROM ReturnToLoading TO Wait_Return := fbDrive.bMoveDone AND tonMoveDelay.Q;
END_TRANSITION
STEP Wait_Return:
	Wait_Return_action(N);
	Wait_Return_exit(P0);
END_STEP
TRANSITION FROM Wait_Return TO Done := tonMoveDelay.Q;
END_TRANSITION
STEP Done:
	Done_action(N);
	Done_exit(P0);
END_STEP
TRANSITION FROM Done TO Init := NOT bExecute;
END_TRANSITION

ACTION Init_exit:
bDone := FALSE;
END_ACTION

ACTION MoveToLow_action:
tonMoveDelay(IN:=TRUE , PT:= tMoveDelay);
fbDrive(
	bEnable:= TRUE,
	bStart:= TRUE,
	wTarget:= GPOS_PIPE_LOW);
END_ACTION

ACTION MoveToLow_exit:
fbDrive(
	bStart:= FALSE);
tonMoveDelay(IN:=FALSE);
END_ACTION

ACTION Wait_Arrive_action:
tonMoveDelay(IN:=TRUE , PT:= tMoveDelay);
END_ACTION

ACTION Wait_Arrive_exit:
tonMoveDelay(IN:=FALSE);
END_ACTION

ACTION Eject_action:
OEjector := TRUE;
tonEjectDelay(IN:=TRUE , PT:= tEjectorDelay);
END_ACTION

ACTION Eject_exit:
tonEjectDelay(IN:=FALSE);
END_ACTION

ACTION ResetEjector_action:
OEjector := FALSE;
tonEjectDelay(IN:=TRUE , PT:= tEjectorDelay);
END_ACTION

ACTION ResetEjector_exit:
tonEjectDelay(IN:=FALSE);
END_ACTION

ACTION ReturnToLoading_action:
fbDrive(
	bEnable:= TRUE,
	bStart:= TRUE,
	wTarget:= GPOS_LOADING);

tonMoveDelay(IN:=TRUE , PT:= tMoveDelay);
END_ACTION

ACTION ReturnToLoading_exit:
fbDrive(
	bStart:= FALSE);

tonMoveDelay(IN:=FALSE);
END_ACTION

ACTION Wait_Return_action:
tonMoveDelay(IN:=TRUE , PT:= tMoveDelay);
END_ACTION

ACTION Wait_Return_exit:
tonMoveDelay(IN:=FALSE);
END_ACTION

ACTION Done_action:
bDone := TRUE;
END_ACTION

ACTION Done_exit:
bDone := FALSE;
END_ACTION
END_PROGRAM

(* POU OLD/PRG_DeliverToMid, SFC *)
PROGRAM PRG_DeliverToMid
VAR_INPUT
	bReset		: BOOL;	(*Reset program*)
	bExecute		: BOOL;	(*enable and run*)
END_VAR
VAR_OUTPUT
	bDone			: BOOL;
END_VAR
VAR
	tonMoveDelay	: TON;
	tonEjectDelay	: TON;
	SFCReset		: BOOL;

	tMoveDelay	: TIME := T#4s;
	tEjectorDelay	: TIME := T#2s;
END_VAR
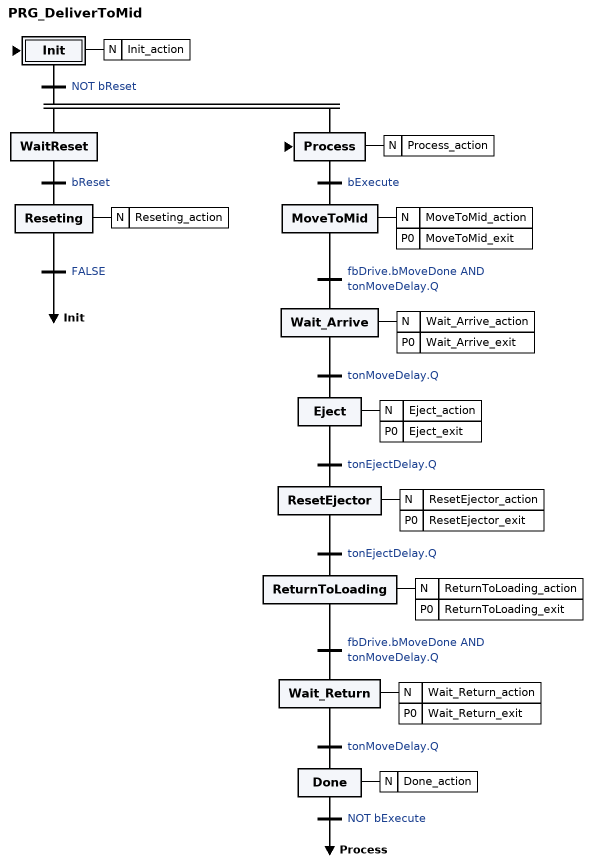
INITIAL_STEP Init:
	Init_action(N);
END_STEP
TRANSITION FROM Init TO (WaitReset, Process) := NOT bReset;
END_TRANSITION
STEP WaitReset:
END_STEP
TRANSITION FROM WaitReset TO Reseting := bReset;
END_TRANSITION
STEP Process:
	Process_action(N);
END_STEP
TRANSITION FROM Process TO MoveToMid := bExecute;
END_TRANSITION
STEP MoveToMid:
	MoveToMid_action(N);
	MoveToMid_exit(P0);
END_STEP
TRANSITION FROM MoveToMid TO Wait_Arrive := fbDrive.bMoveDone AND tonMoveDelay.Q;
END_TRANSITION
STEP Wait_Arrive:
	Wait_Arrive_action(N);
	Wait_Arrive_exit(P0);
END_STEP
TRANSITION FROM Wait_Arrive TO Eject := tonMoveDelay.Q;
END_TRANSITION
STEP Eject:
	Eject_action(N);
	Eject_exit(P0);
END_STEP
TRANSITION FROM Eject TO ResetEjector := tonEjectDelay.Q;
END_TRANSITION
STEP ResetEjector:
	ResetEjector_action(N);
	ResetEjector_exit(P0);
END_STEP
TRANSITION FROM ResetEjector TO ReturnToLoading := tonEjectDelay.Q;
END_TRANSITION
STEP ReturnToLoading:
	ReturnToLoading_action(N);
	ReturnToLoading_exit(P0);
END_STEP
TRANSITION FROM ReturnToLoading TO Wait_Return := fbDrive.bMoveDone AND tonMoveDelay.Q;
END_TRANSITION
STEP Wait_Return:
	Wait_Return_action(N);
	Wait_Return_exit(P0);
END_STEP
TRANSITION FROM Wait_Return TO Done := tonMoveDelay.Q;
END_TRANSITION
STEP Done:
	Done_action(N);
END_STEP
TRANSITION FROM Done TO Process := NOT bExecute;
END_TRANSITION
STEP Reseting:
	Reseting_action(N);
END_STEP
TRANSITION FROM Reseting TO Init := FALSE;
END_TRANSITION

ACTION Init_action:
SFCReset := FALSE;
bDone := FALSE;
END_ACTION

ACTION Process_action:
bDone := FALSE;
END_ACTION

ACTION MoveToMid_action:
bDone := FALSE;

fbDrive(
	bEnable:= TRUE,
	bStart:= TRUE,
	wTarget:=GPOS_PIPE_MID);

tonMoveDelay(IN:=TRUE , PT:= tMoveDelay);
END_ACTION

ACTION MoveToMid_exit:
fbDrive(
	bStart:= FALSE);

tonMoveDelay(IN:=FALSE);
END_ACTION

ACTION Wait_Arrive_action:
tonMoveDelay(IN:=TRUE , PT:= tMoveDelay);
END_ACTION

ACTION Wait_Arrive_exit:
tonMoveDelay(IN:=FALSE);
END_ACTION

ACTION Eject_action:
OEjector := TRUE;
tonEjectDelay(IN:=TRUE , PT:= tEjectorDelay);
END_ACTION

ACTION Eject_exit:
tonEjectDelay(IN:=FALSE);
END_ACTION

ACTION ResetEjector_action:
OEjector := FALSE;
tonEjectDelay(IN:=TRUE , PT:= tEjectorDelay);
END_ACTION

ACTION ResetEjector_exit:
tonEjectDelay(IN:=FALSE);
END_ACTION

ACTION ReturnToLoading_action:
fbDrive(
	bEnable:= TRUE,
	bStart:= TRUE,
	wTarget:= GPOS_LOADING);

tonMoveDelay(IN:=TRUE , PT:= tMoveDelay);
END_ACTION

ACTION ReturnToLoading_exit:
fbDrive(
	bStart:= FALSE);

tonMoveDelay(IN:=FALSE);
END_ACTION

ACTION Wait_Return_action:
tonMoveDelay(IN:=TRUE , PT:= tMoveDelay);
END_ACTION

ACTION Wait_Return_exit:
tonMoveDelay(IN:=FALSE);
END_ACTION

ACTION Done_action:
bDone := TRUE;
END_ACTION

ACTION Reseting_action:
SFCReset := TRUE;
END_ACTION
END_PROGRAM

(* POU OLD/PRG_DeliverToMid2, SFC *)
PROGRAM PRG_DeliverToMid2
VAR_INPUT
	bExecute: BOOL;
END_VAR
VAR_INPUT
	bDone: BOOL;
END_VAR
VAR
	tonMoveDelay	: TON;
	tonEjectDelay	: TON;
	tMoveDelay	: TIME := T#3s;
	tEjectorDelay	: TIME := T#3s;
END_VAR
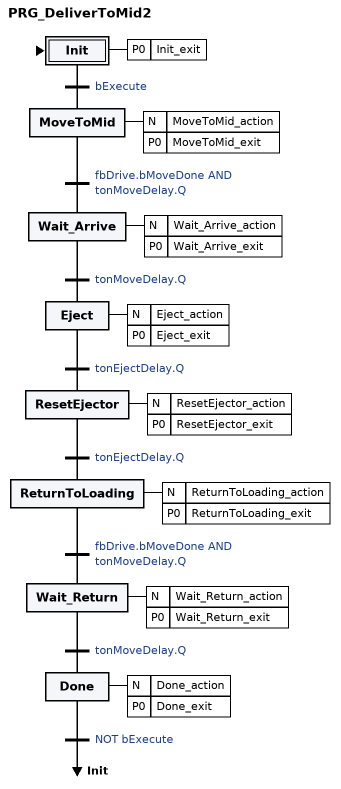
INITIAL_STEP Init:
	Init_exit(P0);
END_STEP
TRANSITION FROM Init TO MoveToMid := bExecute;
END_TRANSITION
STEP MoveToMid:
	MoveToMid_action(N);
	MoveToMid_exit(P0);
END_STEP
TRANSITION FROM MoveToMid TO Wait_Arrive := fbDrive.bMoveDone AND tonMoveDelay.Q;
END_TRANSITION
STEP Wait_Arrive:
	Wait_Arrive_action(N);
	Wait_Arrive_exit(P0);
END_STEP
TRANSITION FROM Wait_Arrive TO Eject := tonMoveDelay.Q;
END_TRANSITION
STEP Eject:
	Eject_action(N);
	Eject_exit(P0);
END_STEP
TRANSITION FROM Eject TO ResetEjector := tonEjectDelay.Q;
END_TRANSITION
STEP ResetEjector:
	ResetEjector_action(N);
	ResetEjector_exit(P0);
END_STEP
TRANSITION FROM ResetEjector TO ReturnToLoading := tonEjectDelay.Q;
END_TRANSITION
STEP ReturnToLoading:
	ReturnToLoading_action(N);
	ReturnToLoading_exit(P0);
END_STEP
TRANSITION FROM ReturnToLoading TO Wait_Return := fbDrive.bMoveDone AND tonMoveDelay.Q;
END_TRANSITION
STEP Wait_Return:
	Wait_Return_action(N);
	Wait_Return_exit(P0);
END_STEP
TRANSITION FROM Wait_Return TO Done := tonMoveDelay.Q;
END_TRANSITION
STEP Done:
	Done_action(N);
	Done_exit(P0);
END_STEP
TRANSITION FROM Done TO Init := NOT bExecute;
END_TRANSITION

ACTION Init_exit:
bDone := FALSE;
END_ACTION

ACTION MoveToMid_action:
fbDrive(
	bEnable:= TRUE,
	bStart:= TRUE,
	wTarget:= GPOS_PIPE_MID);

tonMoveDelay(IN:=TRUE , PT:= tMoveDelay);
END_ACTION

ACTION MoveToMid_exit:
fbDrive(
	bStart:= FALSE);
tonMoveDelay(IN:=FALSE);
END_ACTION

ACTION Wait_Arrive_action:
tonMoveDelay(IN:=TRUE , PT:= tMoveDelay);
END_ACTION

ACTION Wait_Arrive_exit:
tonMoveDelay(IN:=FALSE);
END_ACTION

ACTION Eject_action:
OEjector := TRUE;
tonEjectDelay(IN:=TRUE , PT:= tEjectorDelay);
END_ACTION

ACTION Eject_exit:
tonEjectDelay(IN:=FALSE);
END_ACTION

ACTION ResetEjector_action:
OEjector := FALSE;
tonEjectDelay(IN:=TRUE , PT:= tEjectorDelay);
END_ACTION

ACTION ResetEjector_exit:
tonEjectDelay(IN:=FALSE);
END_ACTION

ACTION ReturnToLoading_action:
fbDrive(
	bEnable:= TRUE,
	bStart:= TRUE,
	wTarget:= GPOS_LOADING);

tonMoveDelay(IN:=TRUE , PT:= tMoveDelay);
END_ACTION

ACTION ReturnToLoading_exit:
fbDrive(
	bStart:= FALSE);

tonMoveDelay(IN:=FALSE);
END_ACTION

ACTION Wait_Return_action:
tonMoveDelay(IN:=TRUE , PT:= tMoveDelay);
END_ACTION

ACTION Wait_Return_exit:
tonMoveDelay(IN:=FALSE);
END_ACTION

ACTION Done_action:
bDone := TRUE;
END_ACTION

ACTION Done_exit:
bDone := FALSE;
END_ACTION
END_PROGRAM

(* POU OLD/PRG_DeliverToUp, SFC *)
PROGRAM PRG_DeliverToUp
VAR_INPUT
	bReset		: BOOL;	(*Reset program*)
	bExecute		: BOOL;	(*enable and run*)
END_VAR
VAR_OUTPUT
	bDone			: BOOL;
END_VAR
VAR
	tonMoveDelay	: TON;
	tonEjectDelay	: TON;
	SFCReset		: BOOL;

	tMoveDelay	: TIME := T#4s;
	tEjectorDelay	: TIME := T#2s;
END_VAR
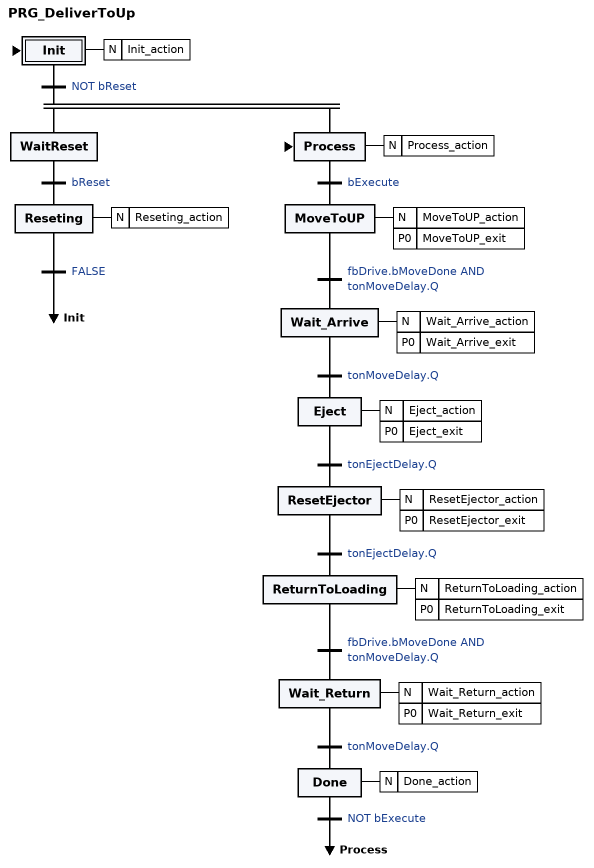
INITIAL_STEP Init:
	Init_action(N);
END_STEP
TRANSITION FROM Init TO (WaitReset, Process) := NOT bReset;
END_TRANSITION
STEP WaitReset:
END_STEP
TRANSITION FROM WaitReset TO Reseting := bReset;
END_TRANSITION
STEP Process:
	Process_action(N);
END_STEP
TRANSITION FROM Process TO MoveToUP := bExecute;
END_TRANSITION
STEP MoveToUP:
	MoveToUP_action(N);
	MoveToUP_exit(P0);
END_STEP
TRANSITION FROM MoveToUP TO Wait_Arrive := fbDrive.bMoveDone AND tonMoveDelay.Q;
END_TRANSITION
STEP Wait_Arrive:
	Wait_Arrive_action(N);
	Wait_Arrive_exit(P0);
END_STEP
TRANSITION FROM Wait_Arrive TO Eject := tonMoveDelay.Q;
END_TRANSITION
STEP Eject:
	Eject_action(N);
	Eject_exit(P0);
END_STEP
TRANSITION FROM Eject TO ResetEjector := tonEjectDelay.Q;
END_TRANSITION
STEP ResetEjector:
	ResetEjector_action(N);
	ResetEjector_exit(P0);
END_STEP
TRANSITION FROM ResetEjector TO ReturnToLoading := tonEjectDelay.Q;
END_TRANSITION
STEP ReturnToLoading:
	ReturnToLoading_action(N);
	ReturnToLoading_exit(P0);
END_STEP
TRANSITION FROM ReturnToLoading TO Wait_Return := fbDrive.bMoveDone AND tonMoveDelay.Q;
END_TRANSITION
STEP Wait_Return:
	Wait_Return_action(N);
	Wait_Return_exit(P0);
END_STEP
TRANSITION FROM Wait_Return TO Done := tonMoveDelay.Q;
END_TRANSITION
STEP Done:
	Done_action(N);
END_STEP
TRANSITION FROM Done TO Process := NOT bExecute;
END_TRANSITION
STEP Reseting:
	Reseting_action(N);
END_STEP
TRANSITION FROM Reseting TO Init := FALSE;
END_TRANSITION

ACTION Init_action:
SFCReset := FALSE;
bDone := FALSE;
END_ACTION

ACTION Process_action:
bDone := FALSE;
END_ACTION

ACTION MoveToUP_action:
bDone := FALSE;

fbDrive(
	bEnable:= TRUE,
	bStart:= TRUE,
	wTarget:= GPOS_PIPE_UP);

tonMoveDelay(IN:=TRUE , PT:= tMoveDelay);
END_ACTION

ACTION MoveToUP_exit:
fbDrive(
	bStart:= FALSE);

tonMoveDelay(IN:=FALSE);
END_ACTION

ACTION Wait_Arrive_action:
tonMoveDelay(IN:=TRUE , PT:= tMoveDelay);
END_ACTION

ACTION Wait_Arrive_exit:
tonMoveDelay(IN:=FALSE);
END_ACTION

ACTION Eject_action:
OEjector := TRUE;
tonEjectDelay(IN:=TRUE , PT:= tEjectorDelay);
END_ACTION

ACTION Eject_exit:
tonEjectDelay(IN:=FALSE);
END_ACTION

ACTION ResetEjector_action:
OEjector := FALSE;
tonEjectDelay(IN:=TRUE , PT:= tEjectorDelay);
END_ACTION

ACTION ResetEjector_exit:
tonEjectDelay(IN:=FALSE);
END_ACTION

ACTION ReturnToLoading_action:
fbDrive(
	bEnable:= TRUE,
	bStart:= TRUE,
	wTarget:= GPOS_LOADING);

tonMoveDelay(IN:=TRUE , PT:= tMoveDelay);
END_ACTION

ACTION ReturnToLoading_exit:
fbDrive(
	bStart:= FALSE);

tonMoveDelay(IN:=FALSE);
END_ACTION

ACTION Wait_Return_action:
tonMoveDelay(IN:=TRUE , PT:= tMoveDelay);
END_ACTION

ACTION Wait_Return_exit:
tonMoveDelay(IN:=FALSE);
END_ACTION

ACTION Done_action:
bDone := TRUE;
END_ACTION

ACTION Reseting_action:
SFCReset := TRUE;
END_ACTION
END_PROGRAM

(* POU OLD/PRG_DeliverToUp2, SFC *)
PROGRAM PRG_DeliverToUp2
VAR_INPUT
	bExecute: BOOL;
END_VAR
VAR_INPUT
	bDone: BOOL;
END_VAR
VAR
	tonMoveDelay	: TON;
	tonEjectDelay	: TON;
	tMoveDelay	: TIME := T#3s;
	tEjectorDelay	: TIME := T#3s;
END_VAR
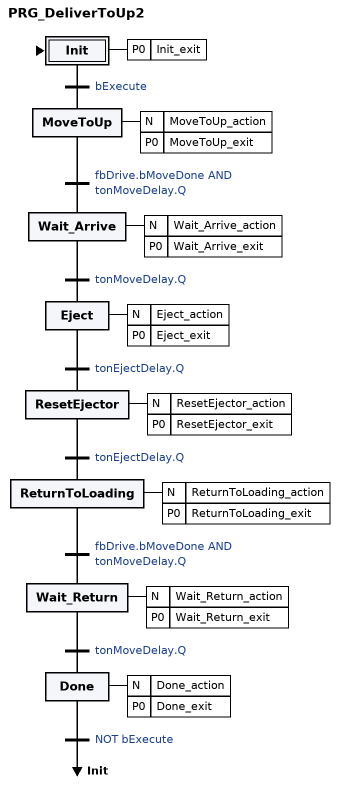
INITIAL_STEP Init:
	Init_exit(P0);
END_STEP
TRANSITION FROM Init TO MoveToUp := bExecute;
END_TRANSITION
STEP MoveToUp:
	MoveToUp_action(N);
	MoveToUp_exit(P0);
END_STEP
TRANSITION FROM MoveToUp TO Wait_Arrive := fbDrive.bMoveDone AND tonMoveDelay.Q;
END_TRANSITION
STEP Wait_Arrive:
	Wait_Arrive_action(N);
	Wait_Arrive_exit(P0);
END_STEP
TRANSITION FROM Wait_Arrive TO Eject := tonMoveDelay.Q;
END_TRANSITION
STEP Eject:
	Eject_action(N);
	Eject_exit(P0);
END_STEP
TRANSITION FROM Eject TO ResetEjector := tonEjectDelay.Q;
END_TRANSITION
STEP ResetEjector:
	ResetEjector_action(N);
	ResetEjector_exit(P0);
END_STEP
TRANSITION FROM ResetEjector TO ReturnToLoading := tonEjectDelay.Q;
END_TRANSITION
STEP ReturnToLoading:
	ReturnToLoading_action(N);
	ReturnToLoading_exit(P0);
END_STEP
TRANSITION FROM ReturnToLoading TO Wait_Return := fbDrive.bMoveDone AND tonMoveDelay.Q;
END_TRANSITION
STEP Wait_Return:
	Wait_Return_action(N);
	Wait_Return_exit(P0);
END_STEP
TRANSITION FROM Wait_Return TO Done := tonMoveDelay.Q;
END_TRANSITION
STEP Done:
	Done_action(N);
	Done_exit(P0);
END_STEP
TRANSITION FROM Done TO Init := NOT bExecute;
END_TRANSITION

ACTION Init_exit:
bDone := FALSE;
END_ACTION

ACTION MoveToUp_action:
fbDrive(
	bEnable:= TRUE,
	bStart:= TRUE,
	wTarget:= GPOS_PIPE_UP);

tonMoveDelay(IN:=TRUE , PT:= tMoveDelay);
END_ACTION

ACTION MoveToUp_exit:
fbDrive(
	bStart:= FALSE);
tonMoveDelay(IN:=FALSE);
END_ACTION

ACTION Wait_Arrive_action:
tonMoveDelay(IN:=TRUE , PT:= tMoveDelay);
END_ACTION

ACTION Wait_Arrive_exit:
tonMoveDelay(IN:=FALSE);
END_ACTION

ACTION Eject_action:
OEjector := TRUE;
tonEjectDelay(IN:=TRUE , PT:= tEjectorDelay);
END_ACTION

ACTION Eject_exit:
tonEjectDelay(IN:=FALSE);
END_ACTION

ACTION ResetEjector_action:
OEjector := FALSE;
tonEjectDelay(IN:=TRUE , PT:= tEjectorDelay);
END_ACTION

ACTION ResetEjector_exit:
tonEjectDelay(IN:=FALSE);
END_ACTION

ACTION ReturnToLoading_action:
fbDrive(
	bEnable:= TRUE,
	bStart:= TRUE,
	wTarget:= GPOS_LOADING);

tonMoveDelay(IN:=TRUE , PT:= tMoveDelay);
END_ACTION

ACTION ReturnToLoading_exit:
fbDrive(
	bStart:= FALSE);

tonMoveDelay(IN:=FALSE);
END_ACTION

ACTION Wait_Return_action:
tonMoveDelay(IN:=TRUE , PT:= tMoveDelay);
END_ACTION

ACTION Wait_Return_exit:
tonMoveDelay(IN:=FALSE);
END_ACTION

ACTION Done_action:
bDone := TRUE;
END_ACTION

ACTION Done_exit:
bDone := FALSE;
END_ACTION
END_PROGRAM

(* POU OLD/PRG_Emptying, ST *)
PROGRAM PRG_Emptying
VAR_INPUT
	bExecute		: BOOL;			(* Execture Auto Sorting Program *)
	bReset			: BOOL := FALSE;(* Reset Program *)
END_VAR
VAR_OUTPUT
	bDone			: BOOL;			(*Program operations done*)
END_VAR
VAR

END_VAR
IF bReset THEN (* Reset Requested *)
	bDone := FALSE;
END_IF
END_PROGRAM

(* POU Processes/PRG_Manual, ST *)
(* This Program performs the automatic sorting of balls into the correct locations.
when the Operator specified batch size has been completed the system enters the 
completing and bDone is Set.  Used in User mode: Sorting
Author: Nicolas Trimborn, nicolas.trimborn@tuni.fi
Date: 	2020-03-01*)

PROGRAM PRG_Manual
VAR_INPUT
	bExecute		: BOOL;			(* Execture Auto Sorting Program *)
	bReset			: BOOL := FALSE;(* Reset Program *)
	iBatchSize  	: INT ;			(* Batch Size to Process *)
END_VAR
VAR_OUTPUT
	bDone			: BOOL;			(*Program operations done*)
	bStopOk			: BOOL;			(*Program is OK to Stop*)
	bBatchComplete  : BOOL;			(*BatchComplete *)
END_VAR
VAR
	iBallsProcessed : INT;			(* Counter for balls Processed *)
	fbSorter		: FB_Sorter;	(* FB implementation for ball sorted lift & gate *)
	fbLift			: FB_Lift;		(* FB implementation for Lift, uses FB_DriveMovement2 *)
END_VAR
actUpdateIO;			(* Updates I/O and calls required function blocks every cycle*)

CASE fbStateModel.eState OF
	eSt_Resetting:
		(*
		IF bBatchComplete THEN
			PRG_HMI.bBtnResetCounters := TRUE;
		END_IF
		*)
		fbStateModel.bSC := TRUE;
	eSt_Stopping: (* Stopping has been requested (HMI or bRun=False *)
		fbStateModel.bStop := FALSE; (* Clear Stop Flag *)

		(* Stop the Sorter and Lift FB, keep executing unitl bStopOk *)
		fbSorter(bEnable:= FALSE, bReset := FALSE);
		fbLift(bEnable:= FALSE, bReset := FALSE);
		IF bStopOk OR NOT bInitCompleted THEN (* System OK to Stop or not initialised*)
			fbStateModel.bSC := TRUE;
		END_IF
	eSt_Execute: (* Execute automatic sorting until batch Completed *)
		IF NOT bBatchComplete THEN
			fbSorter(bEnable := TRUE, bReset := FALSE);
			fbLift(bEnable := TRUE, bReset := FALSE);
		ELSE (*Stop Sorting and trigger Completing State *)
			fbSorter(bEnable := FALSE);
			fbLift(bEnable := FALSE);
			fbStateModel.bComplete := TRUE;
		END_IF

	eSt_Completing: (* Batch Has been Completed *)
		IF bStopOK THEN (* Ensure all FB are ok to stop before entering completed state *)
			bDone := TRUE;
			fbStateModel.bSC := TRUE;
		END_IF

	eSt_Unsuspending: (* Nothing Implemented *)
		fbStateModel.bSC := TRUE;

	eSt_Suspending: (* Nothing Implemented *)
		fbStateModel.bSuspend := FALSE;
		fbStateModel.bSC := TRUE;

END_CASE
END_PROGRAM
ACTION actUpdateIO:
fbSorter (
	I_SensorOpt:= ISensorOpt ,
	I_SensorInd:= ISensorInd,
	I_SorterLiftUp:= ISorterLiftUp ,
	I_SorterLiftDown:= ISorterLiftDown,
	I_SorterGateClosed := ISorterGateClosed,
	hiRdyToReceive_FromDS:= fbLift.hoReadyToRecieve_ToUS ,
	hiBallAvail_FromUS:= ,
	bStopOK=> ,
	bBallLoaded=> ,
	bCurBallMetal=> ,
	O_SorterGate=> OSorterGate ,
	O_SorterLift=> OSorterLift ,
	hoBallAvail_ToDS=> ,
	hoReadyToRecieve_ToUS=> );

fbLift (
	I_LimitUp:= ILimitUp  ,
	I_LimitLow:= ILimitLow,
	I_WaitingBallMetal:= fbSorter.bCurBallMetal  ,
	I_SenColourYellow:= ISenColourYellow ,
	I_SenColourBlue:= ISenColourBlue ,
	I_SenColourGreen:= ISenColourGreen,
	I_SenColourRed:= ISenColourRed ,
	hiRdyToReceive_FromDS:= ,
	hiBallAvail_FromUS:= fbSorter.hoBallAvail_ToDS ,
	bStopOK=> ,
	bBallLoaded=> , 
	bCurBallMetal=> ,
	O_Ejector=> OEjector ,
	hoBallAvail_ToDS=> ,
	hoReadyToRecieve_ToUS=> );

(*
fbPipeUp(
	bReset:= ,
	bEnable:= bExecute,
	I_GateClosed:= IGateClosedUp ,
	I_arrCountBallsIndex:= 3,
	hiRdyToReceive_FromDS:= FALSE ,
	hiBallAvail_FromUS:= ,
	bStopOK=> ,
	bBallLoaded=> ,
	bCurBallMetal=> ,
	O_Gate=> OGateUp,
	hoBallAvail_ToDS=> FALSE ,
	hoReadyToRecieve_ToUS=> );

fbPipeMid(
	bReset:= ,
	bEnable:= bExecute,
	I_GateClosed:= IGateClosedMid,
	I_arrCountBallsIndex:= 2,
	hiRdyToReceive_FromDS:= FALSE ,
	hiBallAvail_FromUS:= ,
	bStopOK=> ,
	bBallLoaded=> ,
	bCurBallMetal=> ,
	O_Gate=> OGateMid,
	hoBallAvail_ToDS=> FALSE,
	hoReadyToRecieve_ToUS=> );

fbPipeLow(
	bReset:= ,
	bEnable:= bExecute,
	I_GateClosed:= IGateClosedLow,
	I_arrCountBallsIndex:= 1,
	hiRdyToReceive_FromDS:= FALSE,
	hiBallAvail_FromUS:= ,
	bStopOK=> ,
	bBallLoaded=> ,
	bCurBallMetal=> ,
	O_Gate=> OGateLow,
	hoBallAvail_ToDS=> FALSE,
	hoReadyToRecieve_ToUS=> );
*)
END_ACTION

(* POU OLD/PRG_MoveToDestOld, SFC *)
PROGRAM PRG_MoveToDestOld
VAR_INPUT
	bExecute: BOOL;
	wTarget : WORD;
END_VAR
VAR_INPUT
	bDone: BOOL;
END_VAR
VAR
	tonMoveDelay	: TON;
	tonEjectDelay	: TON;
	tonSensorDelay	: TON;
	tMoveDelay		: TIME := T#500ms;
	tEjectorDelay	: TIME := T#1s;
	tSensorDelay	: TIME := T#500ms;
END_VAR
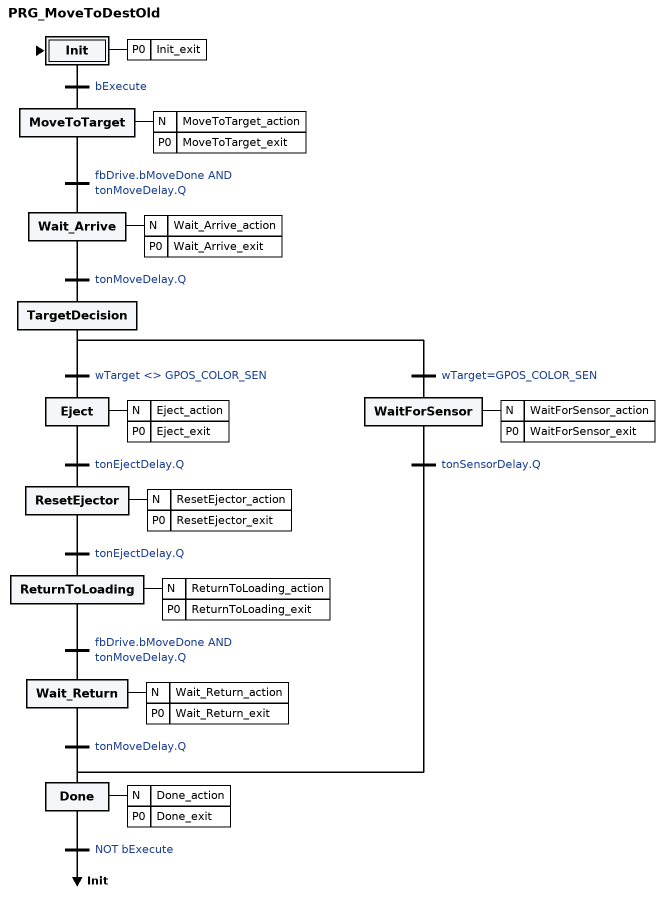
INITIAL_STEP Init:
	Init_exit(P0);
END_STEP
TRANSITION FROM Init TO MoveToTarget := bExecute;
END_TRANSITION
STEP MoveToTarget:
	MoveToTarget_action(N);
	MoveToTarget_exit(P0);
END_STEP
TRANSITION FROM MoveToTarget TO Wait_Arrive := fbDrive.bMoveDone AND tonMoveDelay.Q;
END_TRANSITION
STEP Wait_Arrive:
	Wait_Arrive_action(N);
	Wait_Arrive_exit(P0);
END_STEP
TRANSITION FROM Wait_Arrive TO TargetDecision := tonMoveDelay.Q;
END_TRANSITION
STEP TargetDecision:
END_STEP
TRANSITION FROM TargetDecision TO Eject := wTarget <> GPOS_COLOR_SEN;
END_TRANSITION
TRANSITION FROM TargetDecision TO WaitForSensor := wTarget=GPOS_COLOR_SEN;
END_TRANSITION
STEP WaitForSensor:
	WaitForSensor_action(N);
	WaitForSensor_exit(P0);
END_STEP
TRANSITION FROM WaitForSensor TO Done := tonSensorDelay.Q;
END_TRANSITION
STEP Eject:
	Eject_action(N);
	Eject_exit(P0);
END_STEP
TRANSITION FROM Eject TO ResetEjector := tonEjectDelay.Q;
END_TRANSITION
STEP ResetEjector:
	ResetEjector_action(N);
	ResetEjector_exit(P0);
END_STEP
TRANSITION FROM ResetEjector TO ReturnToLoading := tonEjectDelay.Q;
END_TRANSITION
STEP ReturnToLoading:
	ReturnToLoading_action(N);
	ReturnToLoading_exit(P0);
END_STEP
TRANSITION FROM ReturnToLoading TO Wait_Return := fbDrive.bMoveDone AND tonMoveDelay.Q;
END_TRANSITION
STEP Wait_Return:
	Wait_Return_action(N);
	Wait_Return_exit(P0);
END_STEP
TRANSITION FROM Wait_Return TO Done := tonMoveDelay.Q;
END_TRANSITION
STEP Done:
	Done_action(N);
	Done_exit(P0);
END_STEP
TRANSITION FROM Done TO Init := NOT bExecute;
END_TRANSITION

ACTION Init_exit:
bDone := FALSE;
END_ACTION

ACTION MoveToTarget_action:
tonMoveDelay(IN:=TRUE , PT:= tMoveDelay);
fbDrive(
	bEnable:= TRUE,
	bStart:= TRUE,
	wTarget:= wTarget);
END_ACTION

ACTION MoveToTarget_exit:
fbDrive(
	bStart:= FALSE);
tonMoveDelay(IN:=FALSE);
END_ACTION

ACTION Wait_Arrive_action:
tonMoveDelay(IN:=TRUE , PT:= tMoveDelay);
END_ACTION

ACTION Wait_Arrive_exit:
tonMoveDelay(IN:=FALSE);
END_ACTION

ACTION WaitForSensor_action:
tonSensorDelay(IN:=TRUE , PT:= tSensorDelay);
END_ACTION

ACTION WaitForSensor_exit:
tonSensorDelay(IN:=TRUE , PT:= tSensorDelay);
END_ACTION

ACTION Eject_action:
OEjector := TRUE;
tonEjectDelay(IN:=TRUE , PT:= tEjectorDelay);
END_ACTION

ACTION Eject_exit:
tonEjectDelay(IN:=FALSE);
END_ACTION

ACTION ResetEjector_action:
OEjector := FALSE;
tonEjectDelay(IN:=TRUE , PT:= tEjectorDelay);
END_ACTION

ACTION ResetEjector_exit:
tonEjectDelay(IN:=FALSE);
END_ACTION

ACTION ReturnToLoading_action:
fbDrive(
	bEnable:= TRUE,
	bStart:= TRUE,
	wTarget:= GPOS_LOADING);

tonMoveDelay(IN:=TRUE , PT:= tMoveDelay);
END_ACTION

ACTION ReturnToLoading_exit:
fbDrive(
	bStart:= FALSE);

tonMoveDelay(IN:=FALSE);
END_ACTION

ACTION Wait_Return_action:
tonMoveDelay(IN:=TRUE , PT:= tMoveDelay);
END_ACTION

ACTION Wait_Return_exit:
tonMoveDelay(IN:=FALSE);
END_ACTION

ACTION Done_action:
bDone := TRUE;
END_ACTION

ACTION Done_exit:
bDone := FALSE;
END_ACTION
END_PROGRAM

(* POU OLD/PRG_Sorting_example, SFC *)
PROGRAM PRG_Sorting_example
(*Template program for sorting operation*)
VAR_INPUT
	bReset		: BOOL := FALSE;	(*Reseting the SFC*)
	bExecute	: BOOL;			(*Executes PRG*)
END_VAR
VAR_OUTPUT
	bDone		: BOOL;		(*Program operations done*)
END_VAR
VAR
(* -------------INTERNAL-------------------*)
	bInitDone		: BOOL:=FALSE;	(*Initialisation done*)


(*System variables. See SFC-flags: http://infosys.beckhoff.com/content/1033/tcplccontrol/html/tcplcctrl_editorsfc.htm?id=24319#SFC-Flags*)
	SFCReset		: BOOL := FALSE;	(*For reseting the SFC*)
END_VAR
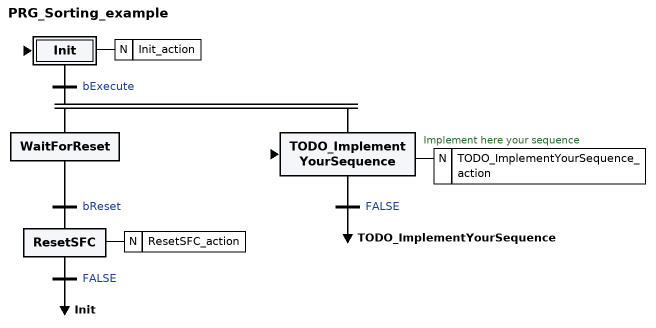
INITIAL_STEP Init:
	Init_action(N);
END_STEP
TRANSITION FROM Init TO (WaitForReset, TODO_ImplementYourSequence) := bExecute;
END_TRANSITION
STEP WaitForReset:
END_STEP
TRANSITION FROM WaitForReset TO ResetSFC := bReset;
END_TRANSITION
STEP TODO_ImplementYourSequence: (* Implement here your sequence *)
	TODO_ImplementYourSequence_action(N);
END_STEP
TRANSITION FROM TODO_ImplementYourSequence TO TODO_ImplementYourSequence := FALSE;
END_TRANSITION
STEP ResetSFC:
	ResetSFC_action(N);
END_STEP
TRANSITION FROM ResetSFC TO Init := FALSE;
END_TRANSITION

ACTION Init_action:
(*Clear Reset SFC*)
SFCReset:= FALSE;
END_ACTION

ACTION TODO_ImplementYourSequence_action:
(*Do some actions...

